LIN {X 0,Y 523.996,Z 356.21,A -85,B 0,C 180,E1 -4869.262,E2 -4869.262} C_VEL
LIN {X 0,Y 523.999,Z 356.208,A -85,B 0,C 180,E1 -4871.743,E2 -4871.743} C_VEL
LIN {X 0,Y 523.985,Z 356.213,A -85,B 0,C 180,E1 -4875.053,E2 -4875.053} C_VEL
LIN {X 0,Y 523.956,Z 356.215,A -85,B 0,C 180,E1 -4877.97,E2 -4877.97} C_VEL
LIN {X 0,Y 523.965,Z 356.22,A -85,B 0,C 180,E1 -4880.411,E2 -4880.411} C_VEL
LIN {X 0,Y 523.909,Z 356.222,A -85,B 0,C 180,E1 -4882.894,E2 -4882.894} C_VEL
LIN {X 0,Y 523.948,Z 356.211,A -85,B 0,C 180,E1 -4885.419,E2 -4885.419} C_VEL
LIN {X 0,Y 523.964,Z 356.214,A -85,B 0,C 180,E1 -4888,E2 -4888} C_VEL
LIN {X 0,Y 523.941,Z 356.216,A -85,B 0,C 180,E1 -4890.856,E2 -4890.856} C_VEL
LIN {X 0,Y 523.956,Z 356.217,A -85,B 0,C 180,E1 -4893.736,E2 -4893.736} C_VEL
LIN {X 0,Y 523.918,Z 356.224,A -85,B 0,C 180,E1 -4896.405,E2 -4896.405} C_VEL
LIN {X 0,Y 523.928,Z 356.218,A -85,B 0,C 180,E1 -4899.085,E2 -4899.085} C_VEL
LIN {X 0,Y 523.955,Z 356.22,A -85,B 0,C 180,E1 -4902.119,E2 -4902.119} C_VEL
LIN {X 0,Y 523.954,Z 356.218,A -85,B 0,C 180,E1 -4905.31,E2 -4905.31} C_VEL
LIN {X 0,Y 523.917,Z 356.22,A -85,B 0,C 180,E1 -4906.929,E2 -4906.929} C_VEL
LIN {X 0,Y 523.255,Z 356.309,A -85,B 0,C 180,E1 -4907.571,E2 -4907.571} C_VEL
LIN {X 0,Y 520.421,Z 356.663,A -85,B 0,C 180,E1 -4908.613,E2 -4908.613} C_VEL
LIN {X 0,Y 518.025,Z 356.962,A -85,B 0,C 180,E1 -4909.452,E2 -4909.452} C_VEL
LIN {X 0,Y 516.995,Z 357.088,A -85,B 0,C 180,E1 -4910.1,E2 -4910.1} C_VEL
LIN {X 0,Y 516.91,Z 357.096,A -85,B 0,C 180,E1 -4910.319,E2 -4910.319} C_VEL
LIN {X 0,Y 516.886,Z 357.099,A -85,B 0,C 180,E1 -4913.343,E2 -4913.343} C_VEL
LIN {X 0,Y 516.914,Z 357.096,A -85,B 0,C 180,E1 -4916.122,E2 -4916.122} C_VEL
LIN {X 0,Y 516.895,Z 357.097,A -85,B 0,C 180,E1 -4918.936,E2 -4918.936} C_VEL
LIN {X 0,Y 516.964,Z 357.229,A -85,B 0,C 180,E1 -4921.72,E2 -4921.72} C_VEL
LIN {X 0,Y 517.544,Z 361.865,A -85,B 0,C 180,E1 -4922.723,E2 -4922.723} C_VEL
LIN {X 0,Y 517.255,Z 376.152,A -85,B 0,C 180,E1 -4925.684,E2 -4925.684} C_VEL
LIN {X 0,Y 519.157,Z 386.668,A -85,B 0,C 180,E1 -4925.908,E2 -4925.908} C_VEL
LIN {X 0,Y 518.645,Z 483.005,A -85,B 0,C 180,E1 -4927.268,E2 -4927.268} C_VEL
LIN {X 0,Y 518.448,Z 496.309,A -85,B 0,C 180,E1 -4927.622,E2 -4927.622} C_VEL
LIN {X 0,Y 518.206,Z 508.549,A -85,B 0,C 180,E1 -4928.102,E2 -4928.102} C_VEL
LIN {X 0,Y 517.961,Z 520.129,A -85,B 0,C 180,E1 -4928.718,E2 -4928.718} C_VEL
LIN {X 0,Y 517.632,Z 531.892,A -85,B 0,C 180,E1 -4929.527,E2 -4929.527} C_VEL
LIN {X 0,Y 517.298,Z 542.625,A -85,B 0,C 180,E1 -4930.455,E2 -4930.455} C_VEL
LIN {X 0,Y 517.062,Z 551.21,A -85,B 0,C 180,E1 -4931.373,E2 -4931.373} C_VEL
LIN {X 0,Y 516.772,Z 560.444,A -85,B 0,C 180,E1 -4932.591,E2 -4932.591} C_VEL
LIN {X 0,Y 516.587,Z 567.819,A -85,B 0,C 180,E1 -4933.806,E2 -4933.806} C_VEL
LIN {X 0,Y 516.47,Z 573.778,A -85,B 0,C 180,E1 -4935.052,E2 -4935.052} C_VEL
LIN {X 0,Y 516.356,Z 578.16,A -85,B 0,C 180,E1 -4936.221,E2 -4936.221} C_VEL
LIN {X 0,Y 516.293,Z 581.562,A -85,B 0,C 180,E1 -4937.421,E2 -4937.421} C_VEL
LIN {X 0,Y 516.286,Z 583.847,A -85,B 0,C 180,E1 -4938.556,E2 -4938.556} C_VEL
LIN {X 0,Y 516.24,Z 585.354,A -85,B 0,C 180,E1 -4939.806,E2 -4939.806} C_VEL
LIN {X 0,Y 516.231,Z 585.782,A -85,B 0,C 180,E1 -4941.388,E2 -4941.388} C_VEL
LIN {X 0,Y 516.273,Z 585.416,A -85,B 0,C 180,E1 -4942.176,E2 -4942.176} C_VEL
LIN {X 0,Y 516.321,Z 583.816,A -85,B 0,C 180,E1 -4943.546,E2 -4943.546} C_VEL
LIN {X 0,Y 516.321,Z 581.857,A -85,B 0,C 180,E1 -4944.533,E2 -4944.533} C_VEL
LIN {X 0,Y 516.358,Z 578.657,A -85,B 0,C 180,E1 -4945.707,E2 -4945.707} C_VEL
LIN {X 0,Y 516.434,Z 574.411,A -85,B 0,C 180,E1 -4946.88,E2 -4946.88} C_VEL
LIN {X 0,Y 516.56,Z 568.007,A -85,B 0,C 180,E1 -4948.246,E2 -4948.246} C_VEL
LIN {X 0,Y 516.803,Z 560.982,A -85,B 0,C 180,E1 -4949.416,E2 -4949.416} C_VEL
LIN {X 0,Y 517.029,Z 552.275,A -85,B 0,C 180,E1 -4950.584,E2 -4950.584} C_VEL
LIN {X 0,Y 517.302,Z 542.393,A -85,B 0,C 180,E1 -4951.654,E2 -4951.654} C_VEL
LIN {X 0,Y 517.551,Z 532.316,A -85,B 0,C 180,E1 -4952.529,E2 -4952.529} C_VEL
LIN {X 0,Y 517.839,Z 521.167,A -85,B 0,C 180,E1 -4953.307,E2 -4953.307} C_VEL
LIN {X 0,Y 518.093,Z 509.628,A -85,B 0,C 180,E1 -4953.938,E2 -4953.938} C_VEL
LIN {X 0,Y 518.351,Z 497.014,A -85,B 0,C 180,E1 -4954.447,E2 -4954.447} C_VEL
LIN {X 0,Y 518.554,Z 483.6,A -85,B 0,C 180,E1 -4954.81,E2 -4954.81} C_VEL
LIN {X 0,Y 518.792,Z 443.561,A -85,B 0,C 180,E1 -4955.393,E2 -4955.393} C_VEL
LIN {X 0,Y 519.07,Z 385.353,A -85,B 0,C 180,E1 -4956.203,E2 -4956.203} C_VEL
LIN {X 0,Y 517.301,Z 376.098,A -85,B 0,C 180,E1 -4956.408,E2 -4956.408} C_VEL
LIN {X 0,Y 517.525,Z 361.723,A -85,B 0,C 180,E1 -4959.379,E2 -4959.379} C_VEL
LIN {X 0,Y 516.973,Z 357.093,A -85,B 0,C 180,E1 -4960.426,E2 -4960.426} C_VEL
LIN {X 0,Y 516.923,Z 357.092,A -85,B 0,C 180,E1 -4963.363,E2 -4963.363} C_VEL
LIN {X 0,Y 516.908,Z 357.093,A -85,B 0,C 180,E1 -4965.778,E2 -4965.778} C_VEL
LIN {X 0,Y 516.93,Z 357.096,A -85,B 0,C 180,E1 -4968.222,E2 -4968.222} C_VEL
LIN {X 0,Y 516.917,Z 357.094,A -85,B 0,C 180,E1 -4970.701,E2 -4970.701} C_VEL
LIN {X 0,Y 516.916,Z 357.097,A -85,B 0,C 180,E1 -4974.071,E2 -4974.071} C_VEL
LIN {X 0,Y 516.93,Z 357.092,A -85,B 0,C 180,E1 -4976.657,E2 -4976.657} C_VEL
LIN {X 0,Y 516.928,Z 357.092,A -85,B 0,C 180,E1 -4979.526,E2 -4979.526} C_VEL
LIN {X 0,Y 516.899,Z 357.096,A -85,B 0,C 180,E1 -4982.543,E2 -4982.543} C_VEL
LIN {X 0,Y 516.884,Z 357.097,A -85,B 0,C 180,E1 -4985.331,E2 -4985.331} C_VEL
LIN {X 0,Y 516.882,Z 357.102,A -85,B 0,C 180,E1 -4987.942,E2 -4987.942} C_VEL
LIN {X 0,Y 516.883,Z 357.096,A -85,B 0,C 180,E1 -4990.741,E2 -4990.741} C_VEL
LIN {X 0,Y 516.882,Z 357.096,A -85,B 0,C 180,E1 -4992.83,E2 -4992.83} C_VEL
LIN {X 0,Y 516.92,Z 357.092,A -85,B 0,C 180,E1 -4995.009,E2 -4995.009} C_VEL
LIN {X 0,Y 516.92,Z 357.093,A -85,B 0,C 180,E1 -4998.397,E2 -4998.397} C_VEL
LIN {X 0,Y 516.882,Z 357.1,A -85,B 0,C 180,E1 -5001.284,E2 -5001.284} C_VEL
LIN {X 0,Y 516.883,Z 357.099,A -85,B 0,C 180,E1 -5004.22,E2 -5004.22} C_VEL
LIN {X 0,Y 516.892,Z 357.097,A -85,B 0,C 180,E1 -5007.052,E2 -5007.052} C_VEL
LIN {X 0,Y 516.886,Z 357.102,A -85,B 0,C 180,E1 -5009.795,E2 -5009.795} C_VEL
LIN {X 0,Y 516.924,Z 357.092,A -85,B 0,C 180,E1 -5012.467,E2 -5012.467} C_VEL
LIN {X 0,Y 516.907,Z 357.097,A -85,B 0,C 180,E1 -5015.071,E2 -5015.071} C_VEL
LIN {X 0,Y 516.905,Z 357.1,A -85,B 0,C 180,E1 -5017.623,E2 -5017.623} C_VEL
LIN {X 0,Y 516.925,Z 357.092,A -85,B 0,C 180,E1 -5020.129,E2 -5020.129} C_VEL
LIN {X 0,Y 516.924,Z 357.092,A -85,B 0,C 180,E1 -5022.596,E2 -5022.596} C_VEL
LIN {X 0,Y 516.942,Z 357.094,A -85,B 0,C 180,E1 -5025.03,E2 -5025.03} C_VEL
LIN {X 0,Y 516.995,Z 357.083,A -85,B 0,C 180,E1 -5028.234,E2 -5028.234} C_VEL
LIN {X 0,Y 516.964,Z 357.092,A -85,B 0,C 180,E1 -5031.399,E2 -5031.399} C_VEL
LIN {X 0,Y 517.002,Z 357.083,A -85,B 0,C 180,E1 -5033.756,E2 -5033.756} C_VEL
LIN {X 0,Y 517.01,Z 357.086,A -85,B 0,C 180,E1 -5036.883,E2 -5036.883} C_VEL
LIN {X 0,Y 517.075,Z 357.073,A -85,B 0,C 180,E1 -5040,E2 -5040} C_VEL
LIN {X 0,Y 517.01,Z 357.086,A -85,B 0,C 180,E1 -5043.117,E2 -5043.117} C_VEL
LIN {X 0,Y 517.002,Z 357.083,A -85,B 0,C 180,E1 -5046.243,E2 -5046.243} C_VEL
LIN {X 0,Y 516.95,Z 357.09,A -85,B 0,C 180,E1 -5049.389,E2 -5049.389} C_VEL
LIN {X 0,Y 516.974,Z 357.086,A -85,B 0,C 180,E1 -5051.824,E2 -5051.824} C_VEL
LIN {X 0,Y 516.937,Z 357.093,A -85,B 0,C 180,E1 -5055.148,E2 -5055.148} C_VEL
LIN {X 0,Y 516.917,Z 357.095,A -85,B 0,C 180,E1 -5058.222,E2 -5058.222} C_VEL
LIN {X 0,Y 516.906,Z 357.099,A -85,B 0,C 180,E1 -5060.702,E2 -5060.702} C_VEL
LIN {X 0,Y 516.883,Z 357.098,A -85,B 0,C 180,E1 -5063.223,E2 -5063.223} C_VEL
LIN {X 0,Y 516.936,Z 357.094,A -85,B 0,C 180,E1 -5066.197,E2 -5066.197} C_VEL
LIN {X 0,Y 516.914,Z 357.093,A -85,B 0,C 180,E1 -5069.305,E2 -5069.305} C_VEL
LIN {X 0,Y 516.894,Z 357.1,A -85,B 0,C 180,E1 -5072.545,E2 -5072.545} C_VEL
LIN {X 0,Y 516.877,Z 357.097,A -85,B 0,C 180,E1 -5075.333,E2 -5075.333} C_VEL
LIN {X 0,Y 516.876,Z 357.101,A -85,B 0,C 180,E1 -5077.944,E2 -5077.944} C_VEL
LIN {X 0,Y 516.899,Z 357.097,A -85,B 0,C 180,E1 -5080.74,E2 -5080.74} C_VEL
LIN {X 0,Y 516.878,Z 357.101,A -85,B 0,C 180,E1 -5083.904,E2 -5083.904} C_VEL
LIN {X 0,Y 516.878,Z 357.104,A -85,B 0,C 180,E1 -5086.108,E2 -5086.108} C_VEL
LIN {X 0,Y 516.913,Z 357.096,A -85,B 0,C 180,E1 -5088.399,E2 -5088.399} C_VEL
LIN {X 0,Y 516.88,Z 357.096,A -85,B 0,C 180,E1 -5091.285,E2 -5091.285} C_VEL
LIN {X 0,Y 516.889,Z 357.1,A -85,B 0,C 180,E1 -5094.222,E2 -5094.222} C_VEL
LIN {X 0,Y 516.897,Z 357.094,A -85,B 0,C 180,E1 -5097.054,E2 -5097.054} C_VEL
LIN {X 0,Y 516.902,Z 357.1,A -85,B 0,C 180,E1 -5099.798,E2 -5099.798} C_VEL
LIN {X 0,Y 516.929,Z 357.094,A -85,B 0,C 180,E1 -5102.468,E2 -5102.468} C_VEL
LIN {X 0,Y 516.969,Z 357.23,A -85,B 0,C 180,E1 -5104.753,E2 -5104.753} C_VEL
LIN {X 0,Y 518.627,Z 366.071,A -85,B 0,C 180,E1 -5106.226,E2 -5106.226} C_VEL
LIN {X 0,Y 518.217,Z 383.586,A -85,B 0,C 180,E1 -5108.938,E2 -5108.938} C_VEL
LIN {X 0,Y 517.667,Z 405.251,A -85,B 0,C 180,E1 -5112.239,E2 -5112.239} C_VEL
LIN {X 0,Y 517.338,Z 421.391,A -85,B 0,C 180,E1 -5114.634,E2 -5114.634} C_VEL
LIN {X 0,Y 519.105,Z 433.695,A -85,B 0,C 180,E1 -5114.86,E2 -5114.86} C_VEL
LIN {X 0,Y 518.651,Z 529.669,A -85,B 0,C 180,E1 -5116.208,E2 -5116.208} C_VEL
LIN {X 0,Y 518.369,Z 542.982,A -85,B 0,C 180,E1 -5116.55,E2 -5116.55} C_VEL
LIN {X 0,Y 518.065,Z 556.304,A -85,B 0,C 180,E1 -5117.066,E2 -5117.066} C_VEL
LIN {X 0,Y 517.745,Z 568.719,A -85,B 0,C 180,E1 -5117.733,E2 -5117.733} C_VEL
LIN {X 0,Y 517.479,Z 580.42,A -85,B 0,C 180,E1 -5118.544,E2 -5118.544} C_VEL
LIN {X 0,Y 517.163,Z 590.646,A -85,B 0,C 180,E1 -5119.429,E2 -5119.429} C_VEL
LIN {X 0,Y 516.901,Z 599.85,A -85,B 0,C 180,E1 -5120.413,E2 -5120.413} C_VEL
LIN {X 0,Y 516.667,Z 608.821,A -85,B 0,C 180,E1 -5121.592,E2 -5121.592} C_VEL
LIN {X 0,Y 516.509,Z 616.045,A -85,B 0,C 180,E1 -5122.77,E2 -5122.77} C_VEL
LIN {X 0,Y 516.423,Z 622.626,A -85,B 0,C 180,E1 -5124.142,E2 -5124.142} C_VEL
LIN {X 0,Y 516.271,Z 626.976,A -85,B 0,C 180,E1 -5125.315,E2 -5125.315} C_VEL
LIN {X 0,Y 516.37,Z 629.286,A -85,B 0,C 180,E1 -5126.098,E2 -5126.098} C_VEL
LIN {X 0,Y 516.282,Z 631.151,A -85,B 0,C 180,E1 -5126.879,E2 -5126.879} C_VEL
LIN {X 0,Y 516.26,Z 632.552,A -85,B 0,C 180,E1 -5127.659,E2 -5127.659} C_VEL
LIN {X 0,Y 516.16,Z 634.157,A -85,B 0,C 180,E1 -5129.22,E2 -5129.22} C_VEL
LIN {X 0,Y 516.158,Z 634.374,A -85,B 0,C 180,E1 -5130,E2 -5130} C_VEL
LIN {X 0,Y 516.192,Z 633.548,A -85,B 0,C 180,E1 -5131.56,E2 -5131.56} C_VEL
LIN {X 0,Y 516.26,Z 632.551,A -85,B 0,C 180,E1 -5132.341,E2 -5132.341} C_VEL
LIN {X 0,Y 516.282,Z 631.149,A -85,B 0,C 180,E1 -5133.121,E2 -5133.121} C_VEL
LIN {X 0,Y 516.313,Z 628.201,A -85,B 0,C 180,E1 -5134.293,E2 -5134.293} C_VEL
LIN {X 0,Y 516.376,Z 624.212,A -85,B 0,C 180,E1 -5135.467,E2 -5135.467} C_VEL
LIN {X 0,Y 516.474,Z 618.319,A -85,B 0,C 180,E1 -5136.791,E2 -5136.791} C_VEL
LIN {X 0,Y 516.606,Z 611.374,A -85,B 0,C 180,E1 -5138.015,E2 -5138.015} C_VEL
LIN {X 0,Y 516.798,Z 603.059,A -85,B 0,C 180,E1 -5139.194,E2 -5139.194} C_VEL
LIN {X 0,Y 517.056,Z 594.541,A -85,B 0,C 180,E1 -5140.177,E2 -5140.177} C_VEL
LIN {X 0,Y 517.376,Z 584.021,A -85,B 0,C 180,E1 -5141.161,E2 -5141.161} C_VEL
LIN {X 0,Y 517.655,Z 572.813,A -85,B 0,C 180,E1 -5142.004,E2 -5142.004} C_VEL
LIN {X 0,Y 517.958,Z 562.213,A -85,B 0,C 180,E1 -5142.638,E2 -5142.638} C_VEL
LIN {X 0,Y 518.209,Z 550.516,A -85,B 0,C 180,E1 -5143.18,E2 -5143.18} C_VEL
LIN {X 0,Y 518.473,Z 537.963,A -85,B 0,C 180,E1 -5143.597,E2 -5143.597} C_VEL
LIN {X 0,Y 518.684,Z 525.252,A -85,B 0,C 180,E1 -5143.866,E2 -5143.866} C_VEL
LIN {X 0,Y 518.996,Z 432.253,A -85,B 0,C 180,E1 -5145.163,E2 -5145.163} C_VEL
LIN {X 0,Y 517.327,Z 421.066,A -85,B 0,C 180,E1 -5145.377,E2 -5145.377} C_VEL
LIN {X 0,Y 517.765,Z 399.658,A -85,B 0,C 180,E1 -5148.601,E2 -5148.601} C_VEL
LIN {X 0,Y 518.262,Z 380.796,A -85,B 0,C 180,E1 -5151.477,E2 -5151.477} C_VEL
LIN {X 0,Y 518.645,Z 366,A -85,B 0,C 180,E1 -5153.774,E2 -5153.774} C_VEL
LIN {X 0,Y 516.951,Z 357.093,A -85,B 0,C 180,E1 -5155.302,E2 -5155.302} C_VEL
LIN {X 0,Y 516.925,Z 357.096,A -85,B 0,C 180,E1 -5158.414,E2 -5158.414} C_VEL
LIN {X 0,Y 516.891,Z 357.093,A -85,B 0,C 180,E1 -5161.109,E2 -5161.109} C_VEL
LIN {X 0,Y 516.911,Z 357.1,A -85,B 0,C 180,E1 -5163.966,E2 -5163.966} C_VEL
LIN {X 0,Y 516.881,Z 357.097,A -85,B 0,C 180,E1 -5166.745,E2 -5166.745} C_VEL
LIN {X 0,Y 516.879,Z 357.102,A -85,B 0,C 180,E1 -5169.72,E2 -5169.72} C_VEL
LIN {X 0,Y 516.912,Z 357.099,A -85,B 0,C 180,E1 -5171.774,E2 -5171.774} C_VEL
LIN {X 0,Y 516.918,Z 357.09,A -85,B 0,C 180,E1 -5175.009,E2 -5175.009} C_VEL
LIN {X 0,Y 516.917,Z 357.09,A -85,B 0,C 180,E1 -5178.397,E2 -5178.397} C_VEL
LIN {X 0,Y 516.881,Z 357.098,A -85,B 0,C 180,E1 -5181.284,E2 -5181.284} C_VEL
LIN {X 0,Y 516.886,Z 357.095,A -85,B 0,C 180,E1 -5184.221,E2 -5184.221} C_VEL
LIN {X 0,Y 516.892,Z 357.097,A -85,B 0,C 180,E1 -5187.053,E2 -5187.053} C_VEL
LIN {X 0,Y 516.895,Z 357.097,A -85,B 0,C 180,E1 -5189.796,E2 -5189.796} C_VEL
LIN {X 0,Y 516.922,Z 357.09,A -85,B 0,C 180,E1 -5192.467,E2 -5192.467} C_VEL
LIN {X 0,Y 516.906,Z 357.091,A -85,B 0,C 180,E1 -5195.072,E2 -5195.072} C_VEL
LIN {X 0,Y 516.904,Z 357.097,A -85,B 0,C 180,E1 -5197.623,E2 -5197.623} C_VEL
LIN {X 0,Y 516.924,Z 357.089,A -85,B 0,C 180,E1 -5200.13,E2 -5200.13} C_VEL
LIN {X 0,Y 516.923,Z 357.091,A -85,B 0,C 180,E1 -5202.596,E2 -5202.596} C_VEL
LIN {X 0,Y 516.932,Z 357.095,A -85,B 0,C 180,E1 -5205.03,E2 -5205.03} C_VEL
LIN {X 0,Y 516.994,Z 357.081,A -85,B 0,C 180,E1 -5208.234,E2 -5208.234} C_VEL
LIN {X 0,Y 516.965,Z 357.089,A -85,B 0,C 180,E1 -5211.4,E2 -5211.4} C_VEL
LIN {X 0,Y 517.002,Z 357.078,A -85,B 0,C 180,E1 -5213.757,E2 -5213.757} C_VEL
LIN {X 0,Y 517.011,Z 357.088,A -85,B 0,C 180,E1 -5216.883,E2 -5216.883} C_VEL
LIN {X 0,Y 517.075,Z 357.07,A -85,B 0,C 180,E1 -5220,E2 -5220} C_VEL
LIN {X 0,Y 517.01,Z 357.081,A -85,B 0,C 180,E1 -5223.117,E2 -5223.117} C_VEL
LIN {X 0,Y 517.002,Z 357.083,A -85,B 0,C 180,E1 -5226.244,E2 -5226.244} C_VEL
LIN {X 0,Y 516.95,Z 357.087,A -85,B 0,C 180,E1 -5229.39,E2 -5229.39} C_VEL
LIN {X 0,Y 516.948,Z 357.087,A -85,B 0,C 180,E1 -5231.811,E2 -5231.811} C_VEL
LIN {X 0,Y 516.938,Z 357.09,A -85,B 0,C 180,E1 -5235.148,E2 -5235.148} C_VEL
LIN {X 0,Y 516.918,Z 357.094,A -85,B 0,C 180,E1 -5238.223,E2 -5238.223} C_VEL
LIN {X 0,Y 516.905,Z 357.096,A -85,B 0,C 180,E1 -5240.702,E2 -5240.702} C_VEL
LIN {X 0,Y 516.904,Z 357.097,A -85,B 0,C 180,E1 -5244.073,E2 -5244.073} C_VEL
LIN {X 0,Y 516.922,Z 357.09,A -85,B 0,C 180,E1 -5246.658,E2 -5246.658} C_VEL
LIN {X 0,Y 516.905,Z 357.093,A -85,B 0,C 180,E1 -5249.525,E2 -5249.525} C_VEL
LIN {X 0,Y 516.895,Z 357.098,A -85,B 0,C 180,E1 -5252.545,E2 -5252.545} C_VEL
LIN {X 0,Y 516.878,Z 357.097,A -85,B 0,C 180,E1 -5255.333,E2 -5255.333} C_VEL
LIN {X 0,Y 516.878,Z 357.103,A -85,B 0,C 180,E1 -5257.944,E2 -5257.944} C_VEL
LIN {X 0,Y 516.901,Z 357.095,A -85,B 0,C 180,E1 -5260.741,E2 -5260.741} C_VEL
LIN {X 0,Y 516.88,Z 357.104,A -85,B 0,C 180,E1 -5263.904,E2 -5263.904} C_VEL
LIN {X 0,Y 516.88,Z 357.102,A -85,B 0,C 180,E1 -5266.108,E2 -5266.108} C_VEL
LIN {X 0,Y 516.904,Z 357.096,A -85,B 0,C 180,E1 -5269.261,E2 -5269.261} C_VEL
LIN {X 0,Y 516.91,Z 357.096,A -85,B 0,C 180,E1 -5270.319,E2 -5270.319} C_VEL
LIN {X 0,Y 516.242,Z 357.177,A -85,B 0,C 180,E1 -5270.969,E2 -5270.969} C_VEL
LIN {X 0,Y 513.384,Z 357.538,A -85,B 0,C 180,E1 -5272.025,E2 -5272.025} C_VEL
LIN {X 0,Y 510.965,Z 357.842,A -85,B 0,C 180,E1 -5272.875,E2 -5272.875} C_VEL
LIN {X 0,Y 509.92,Z 357.97,A -85,B 0,C 180,E1 -5273.531,E2 -5273.531} C_VEL
LIN {X 0,Y 509.832,Z 357.979,A -85,B 0,C 180,E1 -5273.753,E2 -5273.753} C_VEL
LIN {X 0,Y 509.864,Z 357.971,A -85,B 0,C 180,E1 -5276.54,E2 -5276.54} C_VEL
LIN {X 0,Y 509.852,Z 357.978,A -85,B 0,C 180,E1 -5279.335,E2 -5279.335} C_VEL
LIN {X 0,Y 509.904,Z 358.006,A -85,B 0,C 180,E1 -5281.549,E2 -5281.549} C_VEL
LIN {X 0,Y 510.582,Z 363.554,A -85,B 0,C 180,E1 -5282.763,E2 -5282.763} C_VEL
LIN {X 0,Y 510.28,Z 376.526,A -85,B 0,C 180,E1 -5285.479,E2 -5285.479} C_VEL
LIN {X 0,Y 512.342,Z 387.866,A -85,B 0,C 180,E1 -5285.714,E2 -5285.714} C_VEL
LIN {X 0,Y 511.762,Z 482.882,A -85,B 0,C 180,E1 -5287.069,E2 -5287.069} C_VEL
LIN {X 0,Y 511.58,Z 495.634,A -85,B 0,C 180,E1 -5287.405,E2 -5287.405} C_VEL
LIN {X 0,Y 511.321,Z 508.278,A -85,B 0,C 180,E1 -5287.898,E2 -5287.898} C_VEL
LIN {X 0,Y 511.046,Z 520.038,A -85,B 0,C 180,E1 -5288.522,E2 -5288.522} C_VEL
LIN {X 0,Y 510.736,Z 530.852,A -85,B 0,C 180,E1 -5289.262,E2 -5289.262} C_VEL
LIN {X 0,Y 510.372,Z 541.584,A -85,B 0,C 180,E1 -5290.179,E2 -5290.179} C_VEL
LIN {X 0,Y 510.109,Z 550.431,A -85,B 0,C 180,E1 -5291.109,E2 -5291.109} C_VEL
LIN {X 0,Y 509.832,Z 558.487,A -85,B 0,C 180,E1 -5292.137,E2 -5292.137} C_VEL
LIN {X 0,Y 509.629,Z 566.3,A -85,B 0,C 180,E1 -5293.373,E2 -5293.373} C_VEL
LIN {X 0,Y 509.46,Z 571.581,A -85,B 0,C 180,E1 -5294.395,E2 -5294.395} C_VEL
LIN {X 0,Y 509.327,Z 576.648,A -85,B 0,C 180,E1 -5295.619,E2 -5295.619} C_VEL
LIN {X 0,Y 509.243,Z 580.53,A -85,B 0,C 180,E1 -5296.838,E2 -5296.838} C_VEL
LIN {X 0,Y 509.212,Z 584.15,A -85,B 0,C 180,E1 -5298.502,E2 -5298.502} C_VEL
LIN {X 0,Y 509.178,Z 585.572,A -85,B 0,C 180,E1 -5299.663,E2 -5299.663} C_VEL
LIN {X 0,Y 509.094,Z 586.073,A -85,B 0,C 180,E1 -5300.465,E2 -5300.465} C_VEL
LIN {X 0,Y 509.177,Z 585.824,A -85,B 0,C 180,E1 -5302.067,E2 -5302.067} C_VEL
LIN {X 0,Y 509.243,Z 584.192,A -85,B 0,C 180,E1 -5303.552,E2 -5303.552} C_VEL
LIN {X 0,Y 509.249,Z 582.466,A -85,B 0,C 180,E1 -5304.456,E2 -5304.456} C_VEL
LIN {X 0,Y 509.28,Z 579.374,A -85,B 0,C 180,E1 -5305.647,E2 -5305.647} C_VEL
LIN {X 0,Y 509.372,Z 575.24,A -85,B 0,C 180,E1 -5306.836,E2 -5306.836} C_VEL
LIN {X 0,Y 509.474,Z 568.968,A -85,B 0,C 180,E1 -5308.221,E2 -5308.221} C_VEL
LIN {X 0,Y 509.749,Z 562.134,A -85,B 0,C 180,E1 -5309.408,E2 -5309.408} C_VEL
LIN {X 0,Y 510.006,Z 553.606,A -85,B 0,C 180,E1 -5310.592,E2 -5310.592} C_VEL
LIN {X 0,Y 510.282,Z 544.894,A -85,B 0,C 180,E1 -5311.578,E2 -5311.578} C_VEL
LIN {X 0,Y 510.533,Z 534.214,A -85,B 0,C 180,E1 -5312.564,E2 -5312.564} C_VEL
LIN {X 0,Y 510.901,Z 523.424,A -85,B 0,C 180,E1 -5313.352,E2 -5313.352} C_VEL
LIN {X 0,Y 511.174,Z 511.41,A -85,B 0,C 180,E1 -5314.04,E2 -5314.04} C_VEL
LIN {X 0,Y 511.43,Z 498.807,A -85,B 0,C 180,E1 -5314.581,E2 -5314.581} C_VEL
LIN {X 0,Y 511.655,Z 486.163,A -85,B 0,C 180,E1 -5314.949,E2 -5314.949} C_VEL
LIN {X 0,Y 511.761,Z 468.451,A -85,B 0,C 180,E1 -5315.245,E2 -5315.245} C_VEL
LIN {X 0,Y 512.267,Z 386.422,A -85,B 0,C 180,E1 -5316.399,E2 -5316.399} C_VEL
LIN {X 0,Y 510.328,Z 376.422,A -85,B 0,C 180,E1 -5316.619,E2 -5316.619} C_VEL
LIN {X 0,Y 510.531,Z 362.613,A -85,B 0,C 180,E1 -5319.508,E2 -5319.508} C_VEL
LIN {X 0,Y 509.92,Z 357.971,A -85,B 0,C 180,E1 -5320.572,E2 -5320.572} C_VEL
LIN {X 0,Y 509.868,Z 357.971,A -85,B 0,C 180,E1 -5323.552,E2 -5323.552} C_VEL
LIN {X 0,Y 509.861,Z 357.975,A -85,B 0,C 180,E1 -5326.002,E2 -5326.002} C_VEL
LIN {X 0,Y 509.871,Z 357.975,A -85,B 0,C 180,E1 -5328.483,E2 -5328.483} C_VEL
LIN {X 0,Y 509.855,Z 357.972,A -85,B 0,C 180,E1 -5331.001,E2 -5331.001} C_VEL
LIN {X 0,Y 509.841,Z 357.974,A -85,B 0,C 180,E1 -5333.562,E2 -5333.562} C_VEL
LIN {X 0,Y 509.915,Z 357.97,A -85,B 0,C 180,E1 -5336.378,E2 -5336.378} C_VEL
LIN {X 0,Y 509.889,Z 357.968,A -85,B 0,C 180,E1 -5338.843,E2 -5338.843} C_VEL
LIN {X 0,Y 509.824,Z 357.978,A -85,B 0,C 180,E1 -5341.589,E2 -5341.589} C_VEL
LIN {X 0,Y 509.855,Z 357.975,A -85,B 0,C 180,E1 -5344.412,E2 -5344.412} C_VEL
LIN {X 0,Y 509.82,Z 357.977,A -85,B 0,C 180,E1 -5347.34,E2 -5347.34} C_VEL
LIN {X 0,Y 509.837,Z 357.977,A -85,B 0,C 180,E1 -5350.381,E2 -5350.381} C_VEL
LIN {X 0,Y 509.822,Z 357.976,A -85,B 0,C 180,E1 -5353.061,E2 -5353.061} C_VEL
LIN {X 0,Y 509.829,Z 357.98,A -85,B 0,C 180,E1 -5355.791,E2 -5355.791} C_VEL
LIN {X 0,Y 509.863,Z 357.972,A -85,B 0,C 180,E1 -5358.575,E2 -5358.575} C_VEL
LIN {X 0,Y 509.848,Z 357.979,A -85,B 0,C 180,E1 -5361.785,E2 -5361.785} C_VEL
LIN {X 0,Y 509.838,Z 357.974,A -85,B 0,C 180,E1 -5364.622,E2 -5364.622} C_VEL
LIN {X 0,Y 509.86,Z 357.976,A -85,B 0,C 180,E1 -5367.48,E2 -5367.48} C_VEL
LIN {X 0,Y 509.852,Z 357.974,A -85,B 0,C 180,E1 -5370.273,E2 -5370.273} C_VEL
LIN {X 0,Y 509.881,Z 357.971,A -85,B 0,C 180,E1 -5372.944,E2 -5372.944} C_VEL
LIN {X 0,Y 509.869,Z 357.976,A -85,B 0,C 180,E1 -5375.574,E2 -5375.574} C_VEL
LIN {X 0,Y 509.842,Z 357.975,A -85,B 0,C 180,E1 -5378.149,E2 -5378.149} C_VEL
LIN {X 0,Y 509.858,Z 357.973,A -85,B 0,C 180,E1 -5380.681,E2 -5380.681} C_VEL
LIN {X 0,Y 509.88,Z 357.974,A -85,B 0,C 180,E1 -5383.174,E2 -5383.174} C_VEL
LIN {X 0,Y 509.865,Z 357.975,A -85,B 0,C 180,E1 -5385.634,E2 -5385.634} C_VEL
LIN {X 0,Y 509.917,Z 357.969,A -85,B 0,C 180,E1 -5388.874,E2 -5388.874} C_VEL
LIN {X 0,Y 509.943,Z 357.962,A -85,B 0,C 180,E1 -5392.078,E2 -5392.078} C_VEL
LIN {X 0,Y 509.976,Z 357.959,A -85,B 0,C 180,E1 -5394.464,E2 -5394.464} C_VEL
LIN {X 0,Y 510.047,Z 357.95,A -85,B 0,C 180,E1 -5397.631,E2 -5397.631} C_VEL
LIN {X 0,Y 510.058,Z 357.952,A -85,B 0,C 180,E1 -5400.789,E2 -5400.789} C_VEL
LIN {X 0,Y 509.953,Z 357.965,A -85,B 0,C 180,E1 -5403.16,E2 -5403.16} C_VEL
LIN {X 0,Y 509.97,Z 357.96,A -85,B 0,C 180,E1 -5406.33,E2 -5406.33} C_VEL
LIN {X 0,Y 509.91,Z 357.971,A -85,B 0,C 180,E1 -5408.72,E2 -5408.72} C_VEL
LIN {X 0,Y 509.942,Z 357.962,A -85,B 0,C 180,E1 -5411.931,E2 -5411.931} C_VEL
LIN {X 0,Y 509.884,Z 357.971,A -85,B 0,C 180,E1 -5415.242,E2 -5415.242} C_VEL
LIN {X 0,Y 509.879,Z 357.97,A -85,B 0,C 180,E1 -5418.001,E2 -5418.001} C_VEL
LIN {X 0,Y 509.849,Z 357.977,A -85,B 0,C 180,E1 -5421.002,E2 -5421.002} C_VEL
LIN {X 0,Y 509.842,Z 357.974,A -85,B 0,C 180,E1 -5423.563,E2 -5423.563} C_VEL
LIN {X 0,Y 509.905,Z 357.973,A -85,B 0,C 180,E1 -5426.38,E2 -5426.38} C_VEL
LIN {X 0,Y 509.87,Z 357.974,A -85,B 0,C 180,E1 -5428.845,E2 -5428.845} C_VEL
LIN {X 0,Y 509.818,Z 357.977,A -85,B 0,C 180,E1 -5431.59,E2 -5431.59} C_VEL
LIN {X 0,Y 509.848,Z 357.978,A -85,B 0,C 180,E1 -5434.414,E2 -5434.414} C_VEL
LIN {X 0,Y 509.814,Z 357.977,A -85,B 0,C 180,E1 -5437.341,E2 -5437.341} C_VEL
LIN {X 0,Y 509.856,Z 357.977,A -85,B 0,C 180,E1 -5440.381,E2 -5440.381} C_VEL
LIN {X 0,Y 509.835,Z 357.974,A -85,B 0,C 180,E1 -5443.065,E2 -5443.065} C_VEL
LIN {X 0,Y 509.826,Z 357.979,A -85,B 0,C 180,E1 -5445.793,E2 -5445.793} C_VEL
LIN {X 0,Y 509.855,Z 357.974,A -85,B 0,C 180,E1 -5448.576,E2 -5448.576} C_VEL
LIN {X 0,Y 509.849,Z 357.977,A -85,B 0,C 180,E1 -5451.787,E2 -5451.787} C_VEL
LIN {X 0,Y 509.845,Z 357.974,A -85,B 0,C 180,E1 -5454.624,E2 -5454.624} C_VEL
LIN {X 0,Y 509.865,Z 357.972,A -85,B 0,C 180,E1 -5457.482,E2 -5457.482} C_VEL
LIN {X 0,Y 509.881,Z 357.973,A -85,B 0,C 180,E1 -5460.27,E2 -5460.27} C_VEL
LIN {X 0,Y 509.886,Z 357.97,A -85,B 0,C 180,E1 -5462.945,E2 -5462.945} C_VEL
LIN {X 0,Y 509.929,Z 358.066,A -85,B 0,C 180,E1 -5464.571,E2 -5464.571} C_VEL
LIN {X 0,Y 511.646,Z 367.113,A -85,B 0,C 180,E1 -5466.096,E2 -5466.096} C_VEL
LIN {X 0,Y 511.449,Z 377.899,A -85,B 0,C 180,E1 -5467.798,E2 -5467.798} C_VEL
LIN {X 0,Y 510.836,Z 398.069,A -85,B 0,C 180,E1 -5470.929,E2 -5470.929} C_VEL
LIN {X 0,Y 510.365,Z 416.852,A -85,B 0,C 180,E1 -5473.809,E2 -5473.809} C_VEL
LIN {X 0,Y 510.321,Z 420.828,A -85,B 0,C 180,E1 -5474.414,E2 -5474.414} C_VEL
LIN {X 0,Y 512.253,Z 435.543,A -85,B 0,C 180,E1 -5474.683,E2 -5474.683} C_VEL
LIN {X 0,Y 511.751,Z 529.318,A -85,B 0,C 180,E1 -5476.018,E2 -5476.018} C_VEL
LIN {X 0,Y 511.454,Z 542.638,A -85,B 0,C 180,E1 -5476.365,E2 -5476.365} C_VEL
LIN {X 0,Y 511.147,Z 555.965,A -85,B 0,C 180,E1 -5476.888,E2 -5476.888} C_VEL
LIN {X 0,Y 510.824,Z 567.693,A -85,B 0,C 180,E1 -5477.52,E2 -5477.52} C_VEL
LIN {X 0,Y 510.516,Z 578.785,A -85,B 0,C 180,E1 -5478.285,E2 -5478.285} C_VEL
LIN {X 0,Y 510.199,Z 589.261,A -85,B 0,C 180,E1 -5479.183,E2 -5479.183} C_VEL
LIN {X 0,Y 509.938,Z 597.83,A -85,B 0,C 180,E1 -5480.08,E2 -5480.08} C_VEL
LIN {X 0,Y 509.682,Z 605.737,A -85,B 0,C 180,E1 -5481.076,E2 -5481.076} C_VEL
LIN {X 0,Y 509.476,Z 613.463,A -85,B 0,C 180,E1 -5482.271,E2 -5482.271} C_VEL
LIN {X 0,Y 509.317,Z 619.722,A -85,B 0,C 180,E1 -5483.474,E2 -5483.474} C_VEL
LIN {X 0,Y 509.243,Z 625.327,A -85,B 0,C 180,E1 -5484.853,E2 -5484.853} C_VEL
LIN {X 0,Y 509.275,Z 628.953,A -85,B 0,C 180,E1 -5486.044,E2 -5486.044} C_VEL
LIN {X 0,Y 509.201,Z 630.819,A -85,B 0,C 180,E1 -5486.835,E2 -5486.835} C_VEL
LIN {X 0,Y 509.189,Z 632.22,A -85,B 0,C 180,E1 -5487.627,E2 -5487.627} C_VEL
LIN {X 0,Y 509.073,Z 633.824,A -85,B 0,C 180,E1 -5489.209,E2 -5489.209} C_VEL
LIN {X 0,Y 509.069,Z 634.04,A -85,B 0,C 180,E1 -5490,E2 -5490} C_VEL
LIN {X 0,Y 509.112,Z 633.214,A -85,B 0,C 180,E1 -5491.582,E2 -5491.582} C_VEL
LIN {X 0,Y 509.189,Z 632.217,A -85,B 0,C 180,E1 -5492.373,E2 -5492.373} C_VEL
LIN {X 0,Y 509.201,Z 630.814,A -85,B 0,C 180,E1 -5493.165,E2 -5493.165} C_VEL
LIN {X 0,Y 509.206,Z 627.864,A -85,B 0,C 180,E1 -5494.353,E2 -5494.353} C_VEL
LIN {X 0,Y 509.294,Z 623.874,A -85,B 0,C 180,E1 -5495.543,E2 -5495.543} C_VEL
LIN {X 0,Y 509.407,Z 617.839,A -85,B 0,C 180,E1 -5496.914,E2 -5496.914} C_VEL
LIN {X 0,Y 509.551,Z 611.032,A -85,B 0,C 180,E1 -5498.127,E2 -5498.127} C_VEL
LIN {X 0,Y 509.753,Z 602.716,A -85,B 0,C 180,E1 -5499.323,E2 -5499.323} C_VEL
LIN {X 0,Y 510.025,Z 594.197,A -85,B 0,C 180,E1 -5500.319,E2 -5500.319} C_VEL
LIN {X 0,Y 510.387,Z 583.675,A -85,B 0,C 180,E1 -5501.316,E2 -5501.316} C_VEL
LIN {X 0,Y 510.665,Z 572.465,A -85,B 0,C 180,E1 -5502.171,E2 -5502.171} C_VEL
LIN {X 0,Y 511.007,Z 561.864,A -85,B 0,C 180,E1 -5502.813,E2 -5502.813} C_VEL
LIN {X 0,Y 511.298,Z 550.164,A -85,B 0,C 180,E1 -5503.361,E2 -5503.361} C_VEL
LIN {X 0,Y 511.574,Z 537.606,A -85,B 0,C 180,E1 -5503.784,E2 -5503.784} C_VEL
LIN {X 0,Y 511.788,Z 524.885,A -85,B 0,C 180,E1 -5504.057,E2 -5504.057} C_VEL
LIN {X 0,Y 512.117,Z 432.764,A -85,B 0,C 180,E1 -5505.36,E2 -5505.36} C_VEL
LIN {X 0,Y 510.289,Z 420.651,A -85,B 0,C 180,E1 -5505.605,E2 -5505.605} C_VEL
LIN {X 0,Y 510.762,Z 400.678,A -85,B 0,C 180,E1 -5508.657,E2 -5508.657} C_VEL
LIN {X 0,Y 511.308,Z 381.857,A -85,B 0,C 180,E1 -5511.572,E2 -5511.572} C_VEL
LIN {X 0,Y 511.671,Z 367.107,A -85,B 0,C 180,E1 -5513.903,E2 -5513.903} C_VEL
LIN {X 0,Y 509.921,Z 357.97,A -85,B 0,C 180,E1 -5515.484,E2 -5515.484} C_VEL
LIN {X 0,Y 509.886,Z 357.969,A -85,B 0,C 180,E1 -5518.843,E2 -5518.843} C_VEL
LIN {X 0,Y 509.826,Z 357.976,A -85,B 0,C 180,E1 -5521.589,E2 -5521.589} C_VEL
LIN {X 0,Y 509.852,Z 357.975,A -85,B 0,C 180,E1 -5524.412,E2 -5524.412} C_VEL
LIN {X 0,Y 509.817,Z 357.978,A -85,B 0,C 180,E1 -5527.34,E2 -5527.34} C_VEL
LIN {X 0,Y 509.835,Z 357.975,A -85,B 0,C 180,E1 -5530.381,E2 -5530.381} C_VEL
LIN {X 0,Y 509.819,Z 357.975,A -85,B 0,C 180,E1 -5533.062,E2 -5533.062} C_VEL
LIN {X 0,Y 509.826,Z 357.98,A -85,B 0,C 180,E1 -5535.792,E2 -5535.792} C_VEL
LIN {X 0,Y 509.86,Z 357.969,A -85,B 0,C 180,E1 -5538.575,E2 -5538.575} C_VEL
LIN {X 0,Y 509.847,Z 357.977,A -85,B 0,C 180,E1 -5541.785,E2 -5541.785} C_VEL
LIN {X 0,Y 509.84,Z 357.972,A -85,B 0,C 180,E1 -5544.623,E2 -5544.623} C_VEL
LIN {X 0,Y 509.859,Z 357.978,A -85,B 0,C 180,E1 -5547.481,E2 -5547.481} C_VEL
LIN {X 0,Y 509.874,Z 357.968,A -85,B 0,C 180,E1 -5550.268,E2 -5550.268} C_VEL
LIN {X 0,Y 509.88,Z 357.97,A -85,B 0,C 180,E1 -5552.944,E2 -5552.944} C_VEL
LIN {X 0,Y 509.867,Z 357.969,A -85,B 0,C 180,E1 -5555.574,E2 -5555.574} C_VEL
LIN {X 0,Y 509.84,Z 357.973,A -85,B 0,C 180,E1 -5558.15,E2 -5558.15} C_VEL
LIN {X 0,Y 509.857,Z 357.971,A -85,B 0,C 180,E1 -5560.681,E2 -5560.681} C_VEL
LIN {X 0,Y 509.879,Z 357.976,A -85,B 0,C 180,E1 -5563.175,E2 -5563.175} C_VEL
LIN {X 0,Y 509.855,Z 357.972,A -85,B 0,C 180,E1 -5565.634,E2 -5565.634} C_VEL
LIN {X 0,Y 509.92,Z 357.968,A -85,B 0,C 180,E1 -5568.875,E2 -5568.875} C_VEL
LIN {X 0,Y 509.943,Z 357.96,A -85,B 0,C 180,E1 -5572.078,E2 -5572.078} C_VEL
LIN {X 0,Y 509.976,Z 357.955,A -85,B 0,C 180,E1 -5574.464,E2 -5574.464} C_VEL
LIN {X 0,Y 510.047,Z 357.946,A -85,B 0,C 180,E1 -5577.631,E2 -5577.631} C_VEL
LIN {X 0,Y 510.058,Z 357.953,A -85,B 0,C 180,E1 -5580.79,E2 -5580.79} C_VEL
LIN {X 0,Y 509.952,Z 357.96,A -85,B 0,C 180,E1 -5583.16,E2 -5583.16} C_VEL
LIN {X 0,Y 509.97,Z 357.96,A -85,B 0,C 180,E1 -5586.33,E2 -5586.33} C_VEL
LIN {X 0,Y 509.911,Z 357.97,A -85,B 0,C 180,E1 -5588.721,E2 -5588.721} C_VEL
LIN {X 0,Y 509.896,Z 357.966,A -85,B 0,C 180,E1 -5591.932,E2 -5591.932} C_VEL
LIN {X 0,Y 509.885,Z 357.968,A -85,B 0,C 180,E1 -5595.242,E2 -5595.242} C_VEL
LIN {X 0,Y 509.88,Z 357.968,A -85,B 0,C 180,E1 -5598.002,E2 -5598.002} C_VEL
LIN {X 0,Y 509.843,Z 357.973,A -85,B 0,C 180,E1 -5601.002,E2 -5601.002} C_VEL
LIN {X 0,Y 509.829,Z 357.974,A -85,B 0,C 180,E1 -5603.564,E2 -5603.564} C_VEL
LIN {X 0,Y 509.907,Z 357.964,A -85,B 0,C 180,E1 -5606.38,E2 -5606.38} C_VEL
LIN {X 0,Y 509.871,Z 357.971,A -85,B 0,C 180,E1 -5608.845,E2 -5608.845} C_VEL
LIN {X 0,Y 509.82,Z 357.975,A -85,B 0,C 180,E1 -5611.591,E2 -5611.591} C_VEL
LIN {X 0,Y 509.849,Z 357.977,A -85,B 0,C 180,E1 -5614.414,E2 -5614.414} C_VEL
LIN {X 0,Y 509.815,Z 357.976,A -85,B 0,C 180,E1 -5617.341,E2 -5617.341} C_VEL
LIN {X 0,Y 509.858,Z 357.976,A -85,B 0,C 180,E1 -5620.381,E2 -5620.381} C_VEL
LIN {X 0,Y 509.837,Z 357.973,A -85,B 0,C 180,E1 -5623.065,E2 -5623.065} C_VEL
LIN {X 0,Y 509.829,Z 357.982,A -85,B 0,C 180,E1 -5625.793,E2 -5625.793} C_VEL
LIN {X 0,Y 509.865,Z 357.973,A -85,B 0,C 180,E1 -5628.577,E2 -5628.577} C_VEL
LIN {X 0,Y 509.859,Z 357.978,A -85,B 0,C 180,E1 -5631.664,E2 -5631.664} C_VEL
LIN {X 0,Y 509.832,Z 357.979,A -85,B 0,C 180,E1 -5633.753,E2 -5633.753} C_VEL
LIN {X 0,Y 509.167,Z 358.06,A -85,B 0,C 180,E1 -5634.413,E2 -5634.413} C_VEL
LIN {X 0,Y 506.349,Z 358.414,A -85,B 0,C 180,E1 -5635.485,E2 -5635.485} C_VEL
LIN {X 0,Y 503.955,Z 358.71,A -85,B 0,C 180,E1 -5636.348,E2 -5636.348} C_VEL
LIN {X 0,Y 502.906,Z 358.839,A -85,B 0,C 180,E1 -5637.015,E2 -5637.015} C_VEL
LIN {X 0,Y 502.809,Z 358.85,A -85,B 0,C 180,E1 -5637.24,E2 -5637.24} C_VEL
LIN {X 0,Y 502.833,Z 358.852,A -85,B 0,C 180,E1 -5640.063,E2 -5640.063} C_VEL
LIN {X 0,Y 502.871,Z 358.939,A -85,B 0,C 180,E1 -5641.402,E2 -5641.402} C_VEL
LIN {X 0,Y 503.633,Z 364.22,A -85,B 0,C 180,E1 -5642.581,E2 -5642.581} C_VEL
LIN {X 0,Y 503.311,Z 376.831,A -85,B 0,C 180,E1 -5645.258,E2 -5645.258} C_VEL
LIN {X 0,Y 505.461,Z 387.84,A -85,B 0,C 180,E1 -5645.494,E2 -5645.494} C_VEL
LIN {X 0,Y 504.896,Z 482.835,A -85,B 0,C 180,E1 -5646.867,E2 -5646.867} C_VEL
LIN {X 0,Y 504.691,Z 495.935,A -85,B 0,C 180,E1 -5647.214,E2 -5647.214} C_VEL
LIN {X 0,Y 504.41,Z 509.178,A -85,B 0,C 180,E1 -5647.741,E2 -5647.741} C_VEL
LIN {X 0,Y 504.149,Z 519.937,A -85,B 0,C 180,E1 -5648.321,E2 -5648.321} C_VEL
LIN {X 0,Y 503.84,Z 530.31,A -85,B 0,C 180,E1 -5649.029,E2 -5649.029} C_VEL
LIN {X 0,Y 503.428,Z 541.635,A -85,B 0,C 180,E1 -5650,E2 -5650} C_VEL
LIN {X 0,Y 503.111,Z 551.439,A -85,B 0,C 180,E1 -5651.048,E2 -5651.048} C_VEL
LIN {X 0,Y 502.791,Z 559.367,A -85,B 0,C 180,E1 -5652.091,E2 -5652.091} C_VEL
LIN {X 0,Y 502.575,Z 567.058,A -85,B 0,C 180,E1 -5653.342,E2 -5653.342} C_VEL
LIN {X 0,Y 502.379,Z 573.179,A -85,B 0,C 180,E1 -5654.586,E2 -5654.586} C_VEL
LIN {X 0,Y 502.24,Z 577.974,A -85,B 0,C 180,E1 -5655.825,E2 -5655.825} C_VEL
LIN {X 0,Y 502.168,Z 581.604,A -85,B 0,C 180,E1 -5657.061,E2 -5657.061} C_VEL
LIN {X 0,Y 502.123,Z 584.468,A -85,B 0,C 180,E1 -5658.455,E2 -5658.455} C_VEL
LIN {X 0,Y 502.084,Z 585.78,A -85,B 0,C 180,E1 -5659.516,E2 -5659.516} C_VEL
LIN {X 0,Y 502.017,Z 586.354,A -85,B 0,C 180,E1 -5660.329,E2 -5660.329} C_VEL
LIN {X 0,Y 502.051,Z 586.5,A -85,B 0,C 180,E1 -5661.142,E2 -5661.142} C_VEL
LIN {X 0,Y 502.098,Z 586.232,A -85,B 0,C 180,E1 -5661.954,E2 -5661.954} C_VEL
LIN {X 0,Y 502.15,Z 584.547,A -85,B 0,C 180,E1 -5663.571,E2 -5663.571} C_VEL
LIN {X 0,Y 502.181,Z 583.074,A -85,B 0,C 180,E1 -5664.378,E2 -5664.378} C_VEL
LIN {X 0,Y 502.204,Z 580.091,A -85,B 0,C 180,E1 -5665.586,E2 -5665.586} C_VEL
LIN {X 0,Y 502.312,Z 576.07,A -85,B 0,C 180,E1 -5666.792,E2 -5666.792} C_VEL
LIN {X 0,Y 502.361,Z 570.92,A -85,B 0,C 180,E1 -5667.996,E2 -5667.996} C_VEL
LIN {X 0,Y 502.655,Z 564.442,A -85,B 0,C 180,E1 -5669.199,E2 -5669.199} C_VEL
LIN {X 0,Y 502.877,Z 556.437,A -85,B 0,C 180,E1 -5670.4,E2 -5670.4} C_VEL
LIN {X 0,Y 503.168,Z 548.269,A -85,B 0,C 180,E1 -5671.401,E2 -5671.401} C_VEL
LIN {X 0,Y 503.479,Z 538.291,A -85,B 0,C 180,E1 -5672.4,E2 -5672.4} C_VEL
LIN {X 0,Y 503.824,Z 527.027,A -85,B 0,C 180,E1 -5673.299,E2 -5673.299} C_VEL
LIN {X 0,Y 504.226,Z 515.959,A -85,B 0,C 180,E1 -5673.996,E2 -5673.996} C_VEL
LIN {X 0,Y 504.434,Z 504.819,A -85,B 0,C 180,E1 -5674.545,E2 -5674.545} C_VEL
LIN {X 0,Y 504.666,Z 492.213,A -85,B 0,C 180,E1 -5674.993,E2 -5674.993} C_VEL
LIN {X 0,Y 504.912,Z 478.863,A -85,B 0,C 180,E1 -5675.291,E2 -5675.291} C_VEL
LIN {X 0,Y 505.471,Z 387.464,A -85,B 0,C 180,E1 -5676.6,E2 -5676.6} C_VEL
LIN {X 0,Y 503.338,Z 376.73,A -85,B 0,C 180,E1 -5676.836,E2 -5676.836} C_VEL
LIN {X 0,Y 503.547,Z 365.386,A -85,B 0,C 180,E1 -5679.236,E2 -5679.236} C_VEL
LIN {X 0,Y 503.048,Z 359.761,A -85,B 0,C 180,E1 -5680.464,E2 -5680.464} C_VEL
LIN {X 0,Y 502.863,Z 358.85,A -85,B 0,C 180,E1 -5680.671,E2 -5680.671} C_VEL
LIN {X 0,Y 502.837,Z 358.85,A -85,B 0,C 180,E1 -5682.922,E2 -5682.922} C_VEL
LIN {X 0,Y 502.854,Z 358.843,A -85,B 0,C 180,E1 -5685.399,E2 -5685.399} C_VEL
LIN {X 0,Y 502.846,Z 358.849,A -85,B 0,C 180,E1 -5688.12,E2 -5688.12} C_VEL
LIN {X 0,Y 502.833,Z 358.851,A -85,B 0,C 180,E1 -5690.535,E2 -5690.535} C_VEL
LIN {X 0,Y 502.801,Z 358.85,A -85,B 0,C 180,E1 -5693.04,E2 -5693.04} C_VEL
LIN {X 0,Y 502.844,Z 358.847,A -85,B 0,C 180,E1 -5695.675,E2 -5695.675} C_VEL
LIN {X 0,Y 502.845,Z 358.85,A -85,B 0,C 180,E1 -5698.372,E2 -5698.372} C_VEL
LIN {X 0,Y 502.796,Z 358.852,A -85,B 0,C 180,E1 -5701.498,E2 -5701.498} C_VEL
LIN {X 0,Y 502.808,Z 358.853,A -85,B 0,C 180,E1 -5704.444,E2 -5704.444} C_VEL
LIN {X 0,Y 502.782,Z 358.853,A -85,B 0,C 180,E1 -5707.177,E2 -5707.177} C_VEL
LIN {X 0,Y 502.787,Z 358.859,A -85,B 0,C 180,E1 -5710.014,E2 -5710.014} C_VEL
LIN {X 0,Y 502.801,Z 358.855,A -85,B 0,C 180,E1 -5712.198,E2 -5712.198} C_VEL
LIN {X 0,Y 502.799,Z 358.854,A -85,B 0,C 180,E1 -5715.467,E2 -5715.467} C_VEL
LIN {X 0,Y 502.832,Z 358.853,A -85,B 0,C 180,E1 -5717.864,E2 -5717.864} C_VEL
LIN {X 0,Y 502.806,Z 358.851,A -85,B 0,C 180,E1 -5721.024,E2 -5721.024} C_VEL
LIN {X 0,Y 502.778,Z 358.856,A -85,B 0,C 180,E1 -5724.167,E2 -5724.167} C_VEL
LIN {X 0,Y 502.828,Z 358.849,A -85,B 0,C 180,E1 -5726.992,E2 -5726.992} C_VEL
LIN {X 0,Y 502.809,Z 358.853,A -85,B 0,C 180,E1 -5730.064,E2 -5730.064} C_VEL
LIN {X 0,Y 502.829,Z 358.848,A -85,B 0,C 180,E1 -5732.533,E2 -5732.533} C_VEL
LIN {X 0,Y 502.824,Z 358.852,A -85,B 0,C 180,E1 -5735.297,E2 -5735.297} C_VEL
LIN {X 0,Y 502.803,Z 358.854,A -85,B 0,C 180,E1 -5737.827,E2 -5737.827} C_VEL
LIN {X 0,Y 502.818,Z 358.849,A -85,B 0,C 180,E1 -5740.4,E2 -5740.4} C_VEL
LIN {X 0,Y 502.829,Z 358.851,A -85,B 0,C 180,E1 -5742.931,E2 -5742.931} C_VEL
LIN {X 0,Y 502.843,Z 358.851,A -85,B 0,C 180,E1 -5745.429,E2 -5745.429} C_VEL
LIN {X 0,Y 502.886,Z 358.843,A -85,B 0,C 180,E1 -5748.717,E2 -5748.717} C_VEL
LIN {X 0,Y 502.894,Z 358.84,A -85,B 0,C 180,E1 -5751.966,E2 -5751.966} C_VEL
LIN {X 0,Y 502.931,Z 358.836,A -85,B 0,C 180,E1 -5754.386,E2 -5754.386} C_VEL
LIN {X 0,Y 503.017,Z 358.827,A -85,B 0,C 180,E1 -5757.598,E2 -5757.598} C_VEL
LIN {X 0,Y 503.017,Z 358.825,A -85,B 0,C 180,E1 -5760,E2 -5760} C_VEL
LIN {X 0,Y 503.017,Z 358.826,A -85,B 0,C 180,E1 -5762.402,E2 -5762.402} C_VEL
LIN {X 0,Y 502.94,Z 358.835,A -85,B 0,C 180,E1 -5765.613,E2 -5765.613} C_VEL
LIN {X 0,Y 502.893,Z 358.84,A -85,B 0,C 180,E1 -5768.033,E2 -5768.033} C_VEL
LIN {X 0,Y 502.886,Z 358.843,A -85,B 0,C 180,E1 -5771.283,E2 -5771.283} C_VEL
LIN {X 0,Y 502.842,Z 358.852,A -85,B 0,C 180,E1 -5774.571,E2 -5774.571} C_VEL
LIN {X 0,Y 502.853,Z 358.845,A -85,B 0,C 180,E1 -5777.907,E2 -5777.907} C_VEL
LIN {X 0,Y 502.822,Z 358.854,A -85,B 0,C 180,E1 -5780.537,E2 -5780.537} C_VEL
LIN {X 0,Y 502.798,Z 358.854,A -85,B 0,C 180,E1 -5783.04,E2 -5783.04} C_VEL
LIN {X 0,Y 502.834,Z 358.847,A -85,B 0,C 180,E1 -5785.676,E2 -5785.676} C_VEL
LIN {X 0,Y 502.833,Z 358.853,A -85,B 0,C 180,E1 -5788.373,E2 -5788.373} C_VEL
LIN {X 0,Y 502.789,Z 358.852,A -85,B 0,C 180,E1 -5791.5,E2 -5791.5} C_VEL
LIN {X 0,Y 502.8,Z 358.856,A -85,B 0,C 180,E1 -5794.445,E2 -5794.445} C_VEL
LIN {X 0,Y 502.775,Z 358.854,A -85,B 0,C 180,E1 -5797.179,E2 -5797.179} C_VEL
LIN {X 0,Y 502.816,Z 358.854,A -85,B 0,C 180,E1 -5800.013,E2 -5800.013} C_VEL
LIN {X 0,Y 502.818,Z 358.855,A -85,B 0,C 180,E1 -5802.203,E2 -5802.203} C_VEL
LIN {X 0,Y 502.796,Z 358.852,A -85,B 0,C 180,E1 -5805.469,E2 -5805.469} C_VEL
LIN {X 0,Y 502.817,Z 358.848,A -85,B 0,C 180,E1 -5808.935,E2 -5808.935} C_VEL
LIN {X 0,Y 502.792,Z 358.858,A -85,B 0,C 180,E1 -5812.047,E2 -5812.047} C_VEL
LIN {X 0,Y 502.808,Z 358.849,A -85,B 0,C 180,E1 -5815.036,E2 -5815.036} C_VEL
LIN {X 0,Y 502.787,Z 358.86,A -85,B 0,C 180,E1 -5817.917,E2 -5817.917} C_VEL
LIN {X 0,Y 502.839,Z 358.847,A -85,B 0,C 180,E1 -5820.714,E2 -5820.714} C_VEL
LIN {X 0,Y 502.862,Z 358.848,A -85,B 0,C 180,E1 -5823.44,E2 -5823.44} C_VEL
LIN {X 0,Y 502.903,Z 358.893,A -85,B 0,C 180,E1 -5824.387,E2 -5824.387} C_VEL
LIN {X 0,Y 504.778,Z 369.47,A -85,B 0,C 180,E1 -5826.187,E2 -5826.187} C_VEL
LIN {X 0,Y 504.212,Z 387.52,A -85,B 0,C 180,E1 -5829.049,E2 -5829.049} C_VEL
LIN {X 0,Y 503.616,Z 408.494,A -85,B 0,C 180,E1 -5832.331,E2 -5832.331} C_VEL
LIN {X 0,Y 503.279,Z 420.566,A -85,B 0,C 180,E1 -5834.192,E2 -5834.192} C_VEL
LIN {X 0,Y 505.4,Z 435.215,A -85,B 0,C 180,E1 -5834.47,E2 -5834.47} C_VEL
LIN {X 0,Y 504.856,Z 528.967,A -85,B 0,C 180,E1 -5835.823,E2 -5835.823} C_VEL
LIN {X 0,Y 504.569,Z 542.295,A -85,B 0,C 180,E1 -5836.175,E2 -5836.175} C_VEL
LIN {X 0,Y 504.216,Z 555.624,A -85,B 0,C 180,E1 -5836.704,E2 -5836.704} C_VEL
LIN {X 0,Y 503.852,Z 568.17,A -85,B 0,C 180,E1 -5837.397,E2 -5837.397} C_VEL
LIN {X 0,Y 503.491,Z 579.745,A -85,B 0,C 180,E1 -5838.221,E2 -5838.221} C_VEL
LIN {X 0,Y 503.166,Z 589.975,A -85,B 0,C 180,E1 -5839.131,E2 -5839.131} C_VEL
LIN {X 0,Y 502.847,Z 599.18,A -85,B 0,C 180,E1 -5840.142,E2 -5840.142} C_VEL
LIN {X 0,Y 502.552,Z 608.152,A -85,B 0,C 180,E1 -5841.354,E2 -5841.354} C_VEL
LIN {X 0,Y 502.349,Z 615.376,A -85,B 0,C 180,E1 -5842.565,E2 -5842.565} C_VEL
LIN {X 0,Y 502.235,Z 620.253,A -85,B 0,C 180,E1 -5843.573,E2 -5843.573} C_VEL
LIN {X 0,Y 502.175,Z 624.995,A -85,B 0,C 180,E1 -5844.781,E2 -5844.781} C_VEL
LIN {X 0,Y 502.164,Z 628.619,A -85,B 0,C 180,E1 -5845.987,E2 -5845.987} C_VEL
LIN {X 0,Y 502.122,Z 630.487,A -85,B 0,C 180,E1 -5846.791,E2 -5846.791} C_VEL
LIN {X 0,Y 502.12,Z 631.889,A -85,B 0,C 180,E1 -5847.594,E2 -5847.594} C_VEL
LIN {X 0,Y 501.99,Z 633.492,A -85,B 0,C 180,E1 -5849.198,E2 -5849.198} C_VEL
LIN {X 0,Y 501.983,Z 633.707,A -85,B 0,C 180,E1 -5850,E2 -5850} C_VEL
LIN {X 0,Y 502.036,Z 632.88,A -85,B 0,C 180,E1 -5851.604,E2 -5851.604} C_VEL
LIN {X 0,Y 502.12,Z 631.883,A -85,B 0,C 180,E1 -5852.406,E2 -5852.406} C_VEL
LIN {X 0,Y 502.122,Z 630.479,A -85,B 0,C 180,E1 -5853.209,E2 -5853.209} C_VEL
LIN {X 0,Y 502.104,Z 627.526,A -85,B 0,C 180,E1 -5854.415,E2 -5854.415} C_VEL
LIN {X 0,Y 502.211,Z 623.536,A -85,B 0,C 180,E1 -5855.622,E2 -5855.622} C_VEL
LIN {X 0,Y 502.333,Z 617.499,A -85,B 0,C 180,E1 -5857.011,E2 -5857.011} C_VEL
LIN {X 0,Y 502.482,Z 610.69,A -85,B 0,C 180,E1 -5858.242,E2 -5858.242} C_VEL
LIN {X 0,Y 502.719,Z 602.373,A -85,B 0,C 180,E1 -5859.454,E2 -5859.454} C_VEL
LIN {X 0,Y 502.994,Z 593.852,A -85,B 0,C 180,E1 -5860.465,E2 -5860.465} C_VEL
LIN {X 0,Y 503.406,Z 583.329,A -85,B 0,C 180,E1 -5861.475,E2 -5861.475} C_VEL
LIN {X 0,Y 503.679,Z 572.116,A -85,B 0,C 180,E1 -5862.343,E2 -5862.343} C_VEL
LIN {X 0,Y 504.058,Z 561.514,A -85,B 0,C 180,E1 -5862.992,E2 -5862.992} C_VEL
LIN {X 0,Y 504.362,Z 549.808,A -85,B 0,C 180,E1 -5863.548,E2 -5863.548} C_VEL
LIN {X 0,Y 504.697,Z 536.331,A -85,B 0,C 180,E1 -5864.001,E2 -5864.001} C_VEL
LIN {X 0,Y 504.92,Z 522.984,A -85,B 0,C 180,E1 -5864.278,E2 -5864.278} C_VEL
LIN {X 0,Y 505.359,Z 434.109,A -85,B 0,C 180,E1 -5865.546,E2 -5865.546} C_VEL
LIN {X 0,Y 503.262,Z 420.314,A -85,B 0,C 180,E1 -5865.827,E2 -5865.827} C_VEL
LIN {X 0,Y 503.792,Z 400.366,A -85,B 0,C 180,E1 -5868.925,E2 -5868.925} C_VEL
LIN {X 0,Y 504.396,Z 381.608,A -85,B 0,C 180,E1 -5871.883,E2 -5871.883} C_VEL
LIN {X 0,Y 504.836,Z 369.573,A -85,B 0,C 180,E1 -5873.81,E2 -5873.81} C_VEL
LIN {X 0,Y 502.895,Z 358.845,A -85,B 0,C 180,E1 -5875.7,E2 -5875.7} C_VEL
LIN {X 0,Y 502.842,Z 358.85,A -85,B 0,C 180,E1 -5878.372,E2 -5878.372} C_VEL
LIN {X 0,Y 502.797,Z 358.851,A -85,B 0,C 180,E1 -5881.499,E2 -5881.499} C_VEL
LIN {X 0,Y 502.805,Z 358.853,A -85,B 0,C 180,E1 -5884.444,E2 -5884.444} C_VEL
LIN {X 0,Y 502.779,Z 358.854,A -85,B 0,C 180,E1 -5887.178,E2 -5887.178} C_VEL
LIN {X 0,Y 502.785,Z 358.857,A -85,B 0,C 180,E1 -5890.014,E2 -5890.014} C_VEL
LIN {X 0,Y 502.799,Z 358.852,A -85,B 0,C 180,E1 -5892.198,E2 -5892.198} C_VEL
LIN {X 0,Y 502.796,Z 358.853,A -85,B 0,C 180,E1 -5895.467,E2 -5895.467} C_VEL
LIN {X 0,Y 502.83,Z 358.851,A -85,B 0,C 180,E1 -5897.864,E2 -5897.864} C_VEL
LIN {X 0,Y 502.804,Z 358.849,A -85,B 0,C 180,E1 -5901.024,E2 -5901.024} C_VEL
LIN {X 0,Y 502.78,Z 358.853,A -85,B 0,C 180,E1 -5904.166,E2 -5904.166} C_VEL
LIN {X 0,Y 502.826,Z 358.848,A -85,B 0,C 180,E1 -5906.993,E2 -5906.993} C_VEL
LIN {X 0,Y 502.823,Z 358.848,A -85,B 0,C 180,E1 -5910.061,E2 -5910.061} C_VEL
LIN {X 0,Y 502.828,Z 358.846,A -85,B 0,C 180,E1 -5912.533,E2 -5912.533} C_VEL
LIN {X 0,Y 502.823,Z 358.844,A -85,B 0,C 180,E1 -5915.297,E2 -5915.297} C_VEL
LIN {X 0,Y 502.802,Z 358.851,A -85,B 0,C 180,E1 -5917.828,E2 -5917.828} C_VEL
LIN {X 0,Y 502.817,Z 358.846,A -85,B 0,C 180,E1 -5920.4,E2 -5920.4} C_VEL
LIN {X 0,Y 502.828,Z 358.851,A -85,B 0,C 180,E1 -5922.932,E2 -5922.932} C_VEL
LIN {X 0,Y 502.836,Z 358.849,A -85,B 0,C 180,E1 -5925.429,E2 -5925.429} C_VEL
LIN {X 0,Y 502.888,Z 358.842,A -85,B 0,C 180,E1 -5928.717,E2 -5928.717} C_VEL
LIN {X 0,Y 502.893,Z 358.838,A -85,B 0,C 180,E1 -5931.967,E2 -5931.967} C_VEL
LIN {X 0,Y 502.931,Z 358.832,A -85,B 0,C 180,E1 -5934.387,E2 -5934.387} C_VEL
LIN {X 0,Y 503.017,Z 358.822,A -85,B 0,C 180,E1 -5937.598,E2 -5937.598} C_VEL
LIN {X 0,Y 503.017,Z 358.822,A -85,B 0,C 180,E1 -5940,E2 -5940} C_VEL
LIN {X 0,Y 503.017,Z 358.826,A -85,B 0,C 180,E1 -5942.402,E2 -5942.402} C_VEL
LIN {X 0,Y 502.931,Z 358.833,A -85,B 0,C 180,E1 -5945.614,E2 -5945.614} C_VEL
LIN {X 0,Y 502.894,Z 358.837,A -85,B 0,C 180,E1 -5948.034,E2 -5948.034} C_VEL
LIN {X 0,Y 502.873,Z 358.841,A -85,B 0,C 180,E1 -5951.284,E2 -5951.284} C_VEL
LIN {X 0,Y 502.843,Z 358.852,A -85,B 0,C 180,E1 -5954.571,E2 -5954.571} C_VEL
LIN {X 0,Y 502.854,Z 358.843,A -85,B 0,C 180,E1 -5957.908,E2 -5957.908} C_VEL
LIN {X 0,Y 502.821,Z 358.852,A -85,B 0,C 180,E1 -5960.537,E2 -5960.537} C_VEL
LIN {X 0,Y 502.789,Z 358.852,A -85,B 0,C 180,E1 -5963.041,E2 -5963.041} C_VEL
LIN {X 0,Y 502.835,Z 358.842,A -85,B 0,C 180,E1 -5965.676,E2 -5965.676} C_VEL
LIN {X 0,Y 502.834,Z 358.851,A -85,B 0,C 180,E1 -5968.373,E2 -5968.373} C_VEL
LIN {X 0,Y 502.791,Z 358.85,A -85,B 0,C 180,E1 -5971.5,E2 -5971.5} C_VEL
LIN {X 0,Y 502.801,Z 358.855,A -85,B 0,C 180,E1 -5974.446,E2 -5974.446} C_VEL
LIN {X 0,Y 502.777,Z 358.853,A -85,B 0,C 180,E1 -5977.179,E2 -5977.179} C_VEL
LIN {X 0,Y 502.819,Z 358.856,A -85,B 0,C 180,E1 -5980.013,E2 -5980.013} C_VEL
LIN {X 0,Y 502.82,Z 358.851,A -85,B 0,C 180,E1 -5982.203,E2 -5982.203} C_VEL
LIN {X 0,Y 502.799,Z 358.855,A -85,B 0,C 180,E1 -5985.469,E2 -5985.469} C_VEL
LIN {X 0,Y 502.826,Z 358.849,A -85,B 0,C 180,E1 -5989.005,E2 -5989.005} C_VEL
LIN {X 0,Y 502.797,Z 358.857,A -85,B 0,C 180,E1 -5992.047,E2 -5992.047} C_VEL
LIN {X 0,Y 502.811,Z 358.851,A -85,B 0,C 180,E1 -5995.036,E2 -5995.036} C_VEL
LIN {X 0,Y 502.809,Z 358.85,A -85,B 0,C 180,E1 -5997.24,E2 -5997.24} C_VEL
LIN {X 0,Y 502.108,Z 358.943,A -85,B 0,C 180,E1 -5997.909,E2 -5997.909} C_VEL
LIN {X 0,Y 499.244,Z 359.297,A -85,B 0,C 180,E1 -5998.995,E2 -5998.995} C_VEL
LIN {X 0,Y 496.859,Z 359.597,A -85,B 0,C 180,E1 -5999.87,E2 -5999.87} C_VEL
LIN {X 0,Y 495.86,Z 359.719,A -85,B 0,C 180,E1 -6000.545,E2 -6000.545} C_VEL
LIN {X 0,Y 495.791,Z 359.727,A -85,B 0,C 180,E1 -6000.774,E2 -6000.774} C_VEL
LIN {X 0,Y 495.842,Z 359.832,A -85,B 0,C 180,E1 -6001.236,E2 -6001.236} C_VEL
LIN {X 0,Y 496.654,Z 364.911,A -85,B 0,C 180,E1 -6002.392,E2 -6002.392} C_VEL
LIN {X 0,Y 496.34,Z 377.12,A -85,B 0,C 180,E1 -6005.018,E2 -6005.018} C_VEL
LIN {X 0,Y 498.689,Z 389.781,A -85,B 0,C 180,E1 -6005.3,E2 -6005.3} C_VEL
LIN {X 0,Y 498.044,Z 483.351,A -85,B 0,C 180,E1 -6006.672,E2 -6006.672} C_VEL
LIN {X 0,Y 497.826,Z 496.266,A -85,B 0,C 180,E1 -6007.019,E2 -6007.019} C_VEL
LIN {X 0,Y 497.539,Z 508.917,A -85,B 0,C 180,E1 -6007.526,E2 -6007.526} C_VEL
LIN {X 0,Y 497.264,Z 519.816,A -85,B 0,C 180,E1 -6008.114,E2 -6008.114} C_VEL
LIN {X 0,Y 496.893,Z 531.099,A -85,B 0,C 180,E1 -6008.895,E2 -6008.895} C_VEL
LIN {X 0,Y 496.491,Z 541.686,A -85,B 0,C 180,E1 -6009.816,E2 -6009.816} C_VEL
LIN {X 0,Y 496.148,Z 550.625,A -85,B 0,C 180,E1 -6010.772,E2 -6010.772} C_VEL
LIN {X 0,Y 495.809,Z 558.782,A -85,B 0,C 180,E1 -6011.83,E2 -6011.83} C_VEL
LIN {X 0,Y 495.55,Z 566.674,A -85,B 0,C 180,E1 -6013.098,E2 -6013.098} C_VEL
LIN {X 0,Y 495.338,Z 572.934,A -85,B 0,C 180,E1 -6014.361,E2 -6014.361} C_VEL
LIN {X 0,Y 495.187,Z 577.855,A -85,B 0,C 180,E1 -6015.619,E2 -6015.619} C_VEL
LIN {X 0,Y 495.09,Z 581.6,A -85,B 0,C 180,E1 -6016.872,E2 -6016.872} C_VEL
LIN {X 0,Y 495.046,Z 584.773,A -85,B 0,C 180,E1 -6018.401,E2 -6018.401} C_VEL
LIN {X 0,Y 494.996,Z 585.988,A -85,B 0,C 180,E1 -6019.364,E2 -6019.364} C_VEL
LIN {X 0,Y 494.96,Z 586.844,A -85,B 0,C 180,E1 -6021.014,E2 -6021.014} C_VEL
LIN {X 0,Y 495,Z 586.641,A -85,B 0,C 180,E1 -6021.838,E2 -6021.838} C_VEL
LIN {X 0,Y 495.079,Z 585.054,A -85,B 0,C 180,E1 -6023.479,E2 -6023.479} C_VEL
LIN {X 0,Y 495.114,Z 583.675,A -85,B 0,C 180,E1 -6024.298,E2 -6024.298} C_VEL
LIN {X 0,Y 495.113,Z 580.787,A -85,B 0,C 180,E1 -6025.522,E2 -6025.522} C_VEL
LIN {X 0,Y 495.254,Z 576.872,A -85,B 0,C 180,E1 -6026.746,E2 -6026.746} C_VEL
LIN {X 0,Y 495.298,Z 571.859,A -85,B 0,C 180,E1 -6027.967,E2 -6027.967} C_VEL
LIN {X 0,Y 495.599,Z 565.533,A -85,B 0,C 180,E1 -6029.187,E2 -6029.187} C_VEL
LIN {X 0,Y 495.836,Z 557.684,A -85,B 0,C 180,E1 -6030.406,E2 -6030.406} C_VEL
LIN {X 0,Y 496.243,Z 547.935,A -85,B 0,C 180,E1 -6031.623,E2 -6031.623} C_VEL
LIN {X 0,Y 496.533,Z 537.762,A -85,B 0,C 180,E1 -6032.637,E2 -6032.637} C_VEL
LIN {X 0,Y 496.937,Z 526.305,A -85,B 0,C 180,E1 -6033.547,E2 -6033.547} C_VEL
LIN {X 0,Y 497.384,Z 514.952,A -85,B 0,C 180,E1 -6034.254,E2 -6034.254} C_VEL
LIN {X 0,Y 497.56,Z 503.315,A -85,B 0,C 180,E1 -6034.811,E2 -6034.811} C_VEL
LIN {X 0,Y 497.862,Z 489.823,A -85,B 0,C 180,E1 -6035.265,E2 -6035.265} C_VEL
LIN {X 0,Y 498.062,Z 477.706,A -85,B 0,C 180,E1 -6035.516,E2 -6035.516} C_VEL
LIN {X 0,Y 498.529,Z 387.422,A -85,B 0,C 180,E1 -6036.826,E2 -6036.826} C_VEL
LIN {X 0,Y 496.337,Z 377.036,A -85,B 0,C 180,E1 -6037.062,E2 -6037.062} C_VEL
LIN {X 0,Y 496.574,Z 366.247,A -85,B 0,C 180,E1 -6039.367,E2 -6039.367} C_VEL
LIN {X 0,Y 495.985,Z 360.608,A -85,B 0,C 180,E1 -6040.615,E2 -6040.615} C_VEL
LIN {X 0,Y 495.829,Z 359.727,A -85,B 0,C 180,E1 -6040.825,E2 -6040.825} C_VEL
LIN {X 0,Y 495.799,Z 359.727,A -85,B 0,C 180,E1 -6043.944,E2 -6043.944} C_VEL
LIN {X 0,Y 495.783,Z 359.731,A -85,B 0,C 180,E1 -6046.469,E2 -6046.469} C_VEL
LIN {X 0,Y 495.788,Z 359.724,A -85,B 0,C 180,E1 -6049.028,E2 -6049.028} C_VEL
LIN {X 0,Y 495.748,Z 359.729,A -85,B 0,C 180,E1 -6051.628,E2 -6051.628} C_VEL
LIN {X 0,Y 495.783,Z 359.725,A -85,B 0,C 180,E1 -6054.873,E2 -6054.873} C_VEL
LIN {X 0,Y 495.817,Z 359.72,A -85,B 0,C 180,E1 -6056.973,E2 -6056.973} C_VEL
LIN {X 0,Y 495.779,Z 359.732,A -85,B 0,C 180,E1 -6060.149,E2 -6060.149} C_VEL
LIN {X 0,Y 495.795,Z 359.724,A -85,B 0,C 180,E1 -6063.244,E2 -6063.244} C_VEL
LIN {X 0,Y 495.73,Z 359.738,A -85,B 0,C 180,E1 -6066.089,E2 -6066.089} C_VEL
LIN {X 0,Y 495.764,Z 359.728,A -85,B 0,C 180,E1 -6068.767,E2 -6068.767} C_VEL
LIN {X 0,Y 495.755,Z 359.733,A -85,B 0,C 180,E1 -6071.78,E2 -6071.78} C_VEL
LIN {X 0,Y 495.747,Z 359.731,A -85,B 0,C 180,E1 -6075.138,E2 -6075.138} C_VEL
LIN {X 0,Y 495.779,Z 359.729,A -85,B 0,C 180,E1 -6078.221,E2 -6078.221} C_VEL
LIN {X 0,Y 495.765,Z 359.73,A -85,B 0,C 180,E1 -6081.23,E2 -6081.23} C_VEL
LIN {X 0,Y 495.75,Z 359.73,A -85,B 0,C 180,E1 -6084.462,E2 -6084.462} C_VEL
LIN {X 0,Y 495.764,Z 359.731,A -85,B 0,C 180,E1 -6087.405,E2 -6087.405} C_VEL
LIN {X 0,Y 495.76,Z 359.729,A -85,B 0,C 180,E1 -6090.253,E2 -6090.253} C_VEL
LIN {X 0,Y 495.827,Z 359.723,A -85,B 0,C 180,E1 -6093.247,E2 -6093.247} C_VEL
LIN {X 0,Y 495.753,Z 359.735,A -85,B 0,C 180,E1 -6095.725,E2 -6095.725} C_VEL
LIN {X 0,Y 495.753,Z 359.73,A -85,B 0,C 180,E1 -6098.371,E2 -6098.371} C_VEL
LIN {X 0,Y 495.777,Z 359.73,A -85,B 0,C 180,E1 -6100.971,E2 -6100.971} C_VEL
LIN {X 0,Y 495.773,Z 359.731,A -85,B 0,C 180,E1 -6103.529,E2 -6103.529} C_VEL
LIN {X 0,Y 495.793,Z 359.725,A -85,B 0,C 180,E1 -6106.055,E2 -6106.055} C_VEL
LIN {X 0,Y 495.867,Z 359.717,A -85,B 0,C 180,E1 -6108.555,E2 -6108.555} C_VEL
LIN {X 0,Y 495.865,Z 359.717,A -85,B 0,C 180,E1 -6111.852,E2 -6111.852} C_VEL
LIN {X 0,Y 495.889,Z 359.713,A -85,B 0,C 180,E1 -6114.306,E2 -6114.306} C_VEL
LIN {X 0,Y 495.986,Z 359.703,A -85,B 0,C 180,E1 -6117.563,E2 -6117.563} C_VEL
LIN {X 0,Y 495.988,Z 359.7,A -85,B 0,C 180,E1 -6120,E2 -6120} C_VEL
LIN {X 0,Y 495.986,Z 359.703,A -85,B 0,C 180,E1 -6122.436,E2 -6122.436} C_VEL
LIN {X 0,Y 495.896,Z 359.712,A -85,B 0,C 180,E1 -6125.693,E2 -6125.693} C_VEL
LIN {X 0,Y 495.865,Z 359.716,A -85,B 0,C 180,E1 -6128.148,E2 -6128.148} C_VEL
LIN {X 0,Y 495.866,Z 359.717,A -85,B 0,C 180,E1 -6131.445,E2 -6131.445} C_VEL
LIN {X 0,Y 495.785,Z 359.729,A -85,B 0,C 180,E1 -6134.783,E2 -6134.783} C_VEL
LIN {X 0,Y 495.78,Z 359.727,A -85,B 0,C 180,E1 -6137.319,E2 -6137.319} C_VEL
LIN {X 0,Y 495.769,Z 359.728,A -85,B 0,C 180,E1 -6139.89,E2 -6139.89} C_VEL
LIN {X 0,Y 495.756,Z 359.732,A -85,B 0,C 180,E1 -6142.863,E2 -6142.863} C_VEL
LIN {X 0,Y 495.792,Z 359.727,A -85,B 0,C 180,E1 -6146.068,E2 -6146.068} C_VEL
LIN {X 0,Y 495.764,Z 359.73,A -85,B 0,C 180,E1 -6148.815,E2 -6148.815} C_VEL
LIN {X 0,Y 495.751,Z 359.73,A -85,B 0,C 180,E1 -6151.727,E2 -6151.727} C_VEL
LIN {X 0,Y 495.77,Z 359.729,A -85,B 0,C 180,E1 -6154.696,E2 -6154.696} C_VEL
LIN {X 0,Y 495.726,Z 359.733,A -85,B 0,C 180,E1 -6157.562,E2 -6157.562} C_VEL
LIN {X 0,Y 495.774,Z 359.728,A -85,B 0,C 180,E1 -6160.699,E2 -6160.699} C_VEL
LIN {X 0,Y 495.73,Z 359.733,A -85,B 0,C 180,E1 -6163.696,E2 -6163.696} C_VEL
LIN {X 0,Y 495.724,Z 359.736,A -85,B 0,C 180,E1 -6166.306,E2 -6166.306} C_VEL
LIN {X 0,Y 495.763,Z 359.727,A -85,B 0,C 180,E1 -6169.301,E2 -6169.301} C_VEL
LIN {X 0,Y 495.729,Z 359.734,A -85,B 0,C 180,E1 -6172.439,E2 -6172.439} C_VEL
LIN {X 0,Y 495.784,Z 359.726,A -85,B 0,C 180,E1 -6175.458,E2 -6175.458} C_VEL
LIN {X 0,Y 495.759,Z 359.729,A -85,B 0,C 180,E1 -6178.365,E2 -6178.365} C_VEL
LIN {X 0,Y 495.79,Z 359.728,A -85,B 0,C 180,E1 -6181.507,E2 -6181.507} C_VEL
LIN {X 0,Y 495.839,Z 359.823,A -85,B 0,C 180,E1 -6184.218,E2 -6184.218} C_VEL
LIN {X 0,Y 497.813,Z 370.584,A -85,B 0,C 180,E1 -6186.076,E2 -6186.076} C_VEL
LIN {X 0,Y 497.267,Z 387.995,A -85,B 0,C 180,E1 -6188.875,E2 -6188.875} C_VEL
LIN {X 0,Y 496.606,Z 409.51,A -85,B 0,C 180,E1 -6192.286,E2 -6192.286} C_VEL
LIN {X 0,Y 496.276,Z 420.238,A -85,B 0,C 180,E1 -6193.964,E2 -6193.964} C_VEL
LIN {X 0,Y 498.556,Z 436.2,A -85,B 0,C 180,E1 -6194.271,E2 -6194.271} C_VEL
LIN {X 0,Y 497.972,Z 528.616,A -85,B 0,C 180,E1 -6195.623,E2 -6195.623} C_VEL
LIN {X 0,Y 497.669,Z 541.95,A -85,B 0,C 180,E1 -6195.979,E2 -6195.979} C_VEL
LIN {X 0,Y 497.284,Z 555.283,A -85,B 0,C 180,E1 -6196.515,E2 -6196.515} C_VEL
LIN {X 0,Y 496.872,Z 567.835,A -85,B 0,C 180,E1 -6197.217,E2 -6197.217} C_VEL
LIN {X 0,Y 496.488,Z 579.407,A -85,B 0,C 180,E1 -6198.052,E2 -6198.052} C_VEL
LIN {X 0,Y 496.17,Z 589.64,A -85,B 0,C 180,E1 -6198.976,E2 -6198.976} C_VEL
LIN {X 0,Y 495.791,Z 598.844,A -85,B 0,C 180,E1 -6200,E2 -6200} C_VEL
LIN {X 0,Y 495.481,Z 607.816,A -85,B 0,C 180,E1 -6201.23,E2 -6201.23} C_VEL
LIN {X 0,Y 495.28,Z 615.042,A -85,B 0,C 180,E1 -6202.458,E2 -6202.458} C_VEL
LIN {X 0,Y 495.124,Z 621.101,A -85,B 0,C 180,E1 -6203.758,E2 -6203.758} C_VEL
LIN {X 0,Y 495.037,Z 625.978,A -85,B 0,C 180,E1 -6205.114,E2 -6205.114} C_VEL
LIN {X 0,Y 495.055,Z 628.286,A -85,B 0,C 180,E1 -6205.93,E2 -6205.93} C_VEL
LIN {X 0,Y 495.045,Z 630.155,A -85,B 0,C 180,E1 -6206.745,E2 -6206.745} C_VEL
LIN {X 0,Y 495.024,Z 631.556,A -85,B 0,C 180,E1 -6207.559,E2 -6207.559} C_VEL
LIN {X 0,Y 494.91,Z 633.159,A -85,B 0,C 180,E1 -6209.186,E2 -6209.186} C_VEL
LIN {X 0,Y 494.901,Z 633.375,A -85,B 0,C 180,E1 -6210,E2 -6210} C_VEL
LIN {X 0,Y 494.963,Z 632.547,A -85,B 0,C 180,E1 -6211.627,E2 -6211.627} C_VEL
LIN {X 0,Y 495.024,Z 631.547,A -85,B 0,C 180,E1 -6212.441,E2 -6212.441} C_VEL
LIN {X 0,Y 495.045,Z 630.144,A -85,B 0,C 180,E1 -6213.255,E2 -6213.255} C_VEL
LIN {X 0,Y 495.009,Z 627.189,A -85,B 0,C 180,E1 -6214.479,E2 -6214.479} C_VEL
LIN {X 0,Y 495.127,Z 623.197,A -85,B 0,C 180,E1 -6215.702,E2 -6215.702} C_VEL
LIN {X 0,Y 495.256,Z 617.057,A -85,B 0,C 180,E1 -6217.133,E2 -6217.133} C_VEL
LIN {X 0,Y 495.428,Z 610.349,A -85,B 0,C 180,E1 -6218.36,E2 -6218.36} C_VEL
LIN {X 0,Y 495.681,Z 602.03,A -85,B 0,C 180,E1 -6219.59,E2 -6219.59} C_VEL
LIN {X 0,Y 495.985,Z 593.507,A -85,B 0,C 180,E1 -6220.615,E2 -6220.615} C_VEL
LIN {X 0,Y 496.425,Z 582.983,A -85,B 0,C 180,E1 -6221.638,E2 -6221.638} C_VEL
LIN {X 0,Y 496.699,Z 572.087,A -85,B 0,C 180,E1 -6222.496,E2 -6222.496} C_VEL
LIN {X 0,Y 497.101,Z 561.162,A -85,B 0,C 180,E1 -6223.178,E2 -6223.178} C_VEL
LIN {X 0,Y 497.439,Z 549.454,A -85,B 0,C 180,E1 -6223.741,E2 -6223.741} C_VEL
LIN {X 0,Y 497.783,Z 536.888,A -85,B 0,C 180,E1 -6224.174,E2 -6224.174} C_VEL
LIN {X 0,Y 498.039,Z 524.148,A -85,B 0,C 180,E1 -6224.453,E2 -6224.453} C_VEL
LIN {X 0,Y 498.485,Z 434.84,A -85,B 0,C 180,E1 -6225.75,E2 -6225.75} C_VEL
LIN {X 0,Y 496.262,Z 420.064,A -85,B 0,C 180,E1 -6226.045,E2 -6226.045} C_VEL
LIN {X 0,Y 496.857,Z 400.088,A -85,B 0,C 180,E1 -6229.2,E2 -6229.2} C_VEL
LIN {X 0,Y 497.462,Z 382.721,A -85,B 0,C 180,E1 -6231.986,E2 -6231.986} C_VEL
LIN {X 0,Y 497.896,Z 370.72,A -85,B 0,C 180,E1 -6233.942,E2 -6233.942} C_VEL
LIN {X 0,Y 495.854,Z 359.723,A -85,B 0,C 180,E1 -6235.894,E2 -6235.894} C_VEL
LIN {X 0,Y 495.78,Z 359.726,A -85,B 0,C 180,E1 -6238.814,E2 -6238.814} C_VEL
LIN {X 0,Y 495.758,Z 359.73,A -85,B 0,C 180,E1 -6241.726,E2 -6241.726} C_VEL
LIN {X 0,Y 495.775,Z 359.727,A -85,B 0,C 180,E1 -6244.695,E2 -6244.695} C_VEL
LIN {X 0,Y 495.729,Z 359.735,A -85,B 0,C 180,E1 -6247.561,E2 -6247.561} C_VEL
LIN {X 0,Y 495.763,Z 359.726,A -85,B 0,C 180,E1 -6250.699,E2 -6250.699} C_VEL
LIN {X 0,Y 495.729,Z 359.734,A -85,B 0,C 180,E1 -6254,E2 -6254} C_VEL
LIN {X 0,Y 495.758,Z 359.727,A -85,B 0,C 180,E1 -6257.12,E2 -6257.12} C_VEL
LIN {X 0,Y 495.777,Z 359.724,A -85,B 0,C 180,E1 -6260.364,E2 -6260.364} C_VEL
LIN {X 0,Y 495.728,Z 359.736,A -85,B 0,C 180,E1 -6263.456,E2 -6263.456} C_VEL
LIN {X 0,Y 495.754,Z 359.727,A -85,B 0,C 180,E1 -6266.435,E2 -6266.435} C_VEL
LIN {X 0,Y 495.75,Z 359.734,A -85,B 0,C 180,E1 -6269.313,E2 -6269.313} C_VEL
LIN {X 0,Y 495.775,Z 359.725,A -85,B 0,C 180,E1 -6272.108,E2 -6272.108} C_VEL
LIN {X 0,Y 495.782,Z 359.719,A -85,B 0,C 180,E1 -6274.832,E2 -6274.832} C_VEL
LIN {X 0,Y 495.752,Z 359.734,A -85,B 0,C 180,E1 -6277.495,E2 -6277.495} C_VEL
LIN {X 0,Y 495.769,Z 359.724,A -85,B 0,C 180,E1 -6280.11,E2 -6280.11} C_VEL
LIN {X 0,Y 495.779,Z 359.726,A -85,B 0,C 180,E1 -6282.681,E2 -6282.681} C_VEL
LIN {X 0,Y 495.781,Z 359.729,A -85,B 0,C 180,E1 -6285.217,E2 -6285.217} C_VEL
LIN {X 0,Y 495.868,Z 359.715,A -85,B 0,C 180,E1 -6288.555,E2 -6288.555} C_VEL
LIN {X 0,Y 495.865,Z 359.714,A -85,B 0,C 180,E1 -6291.852,E2 -6291.852} C_VEL
LIN {X 0,Y 495.888,Z 359.708,A -85,B 0,C 180,E1 -6294.307,E2 -6294.307} C_VEL
LIN {X 0,Y 495.986,Z 359.698,A -85,B 0,C 180,E1 -6297.564,E2 -6297.564} C_VEL
LIN {X 0,Y 495.988,Z 359.697,A -85,B 0,C 180,E1 -6300,E2 -6300} C_VEL
LIN {X 0,Y 495.986,Z 359.702,A -85,B 0,C 180,E1 -6302.437,E2 -6302.437} C_VEL
LIN {X 0,Y 495.889,Z 359.711,A -85,B 0,C 180,E1 -6305.694,E2 -6305.694} C_VEL
LIN {X 0,Y 495.865,Z 359.713,A -85,B 0,C 180,E1 -6308.148,E2 -6308.148} C_VEL
LIN {X 0,Y 495.846,Z 359.715,A -85,B 0,C 180,E1 -6311.446,E2 -6311.446} C_VEL
LIN {X 0,Y 495.786,Z 359.729,A -85,B 0,C 180,E1 -6314.783,E2 -6314.783} C_VEL
LIN {X 0,Y 495.78,Z 359.723,A -85,B 0,C 180,E1 -6317.319,E2 -6317.319} C_VEL
LIN {X 0,Y 495.77,Z 359.727,A -85,B 0,C 180,E1 -6319.891,E2 -6319.891} C_VEL
LIN {X 0,Y 495.751,Z 359.73,A -85,B 0,C 180,E1 -6322.861,E2 -6322.861} C_VEL
LIN {X 0,Y 495.793,Z 359.722,A -85,B 0,C 180,E1 -6326.068,E2 -6326.068} C_VEL
LIN {X 0,Y 495.766,Z 359.728,A -85,B 0,C 180,E1 -6328.816,E2 -6328.816} C_VEL
LIN {X 0,Y 495.753,Z 359.728,A -85,B 0,C 180,E1 -6331.727,E2 -6331.727} C_VEL
LIN {X 0,Y 495.771,Z 359.728,A -85,B 0,C 180,E1 -6334.696,E2 -6334.696} C_VEL
LIN {X 0,Y 495.728,Z 359.733,A -85,B 0,C 180,E1 -6337.562,E2 -6337.562} C_VEL
LIN {X 0,Y 495.777,Z 359.727,A -85,B 0,C 180,E1 -6340.699,E2 -6340.699} C_VEL
LIN {X 0,Y 495.732,Z 359.735,A -85,B 0,C 180,E1 -6343.696,E2 -6343.696} C_VEL
LIN {X 0,Y 495.727,Z 359.736,A -85,B 0,C 180,E1 -6346.306,E2 -6346.306} C_VEL
LIN {X 0,Y 495.78,Z 359.728,A -85,B 0,C 180,E1 -6349.303,E2 -6349.303} C_VEL
LIN {X 0,Y 495.764,Z 359.731,A -85,B 0,C 180,E1 -6351.411,E2 -6351.411} C_VEL
LIN {X 0,Y 495.759,Z 359.729,A -85,B 0,C 180,E1 -6354.464,E2 -6354.464} C_VEL
LIN {X 0,Y 495.77,Z 359.731,A -85,B 0,C 180,E1 -6357.407,E2 -6357.407} C_VEL
LIN {X 0,Y 495.791,Z 359.727,A -85,B 0,C 180,E1 -6360.774,E2 -6360.774} C_VEL
LIN {X 0,Y 495.532,Z 360.389,A -85,B 0,C 180,E1 -6361.225,E2 -6361.225} C_VEL
LIN {X 0,Y 494.385,Z 362.959,A -85,B 0,C 180,E1 -6361.848,E2 -6361.848} C_VEL
LIN {X 0,Y 490.609,Z 370.011,A -85,B 0,C 180,E1 -6363.194,E2 -6363.194} C_VEL
LIN {X 0,Y 489.614,Z 372.898,A -85,B 0,C 180,E1 -6363.792,E2 -6363.792} C_VEL
LIN {X 0,Y 489.507,Z 373.846,A -85,B 0,C 180,E1 -6363.996,E2 -6363.996} C_VEL
LIN {X 0,Y 489.385,Z 377.516,A -85,B 0,C 180,E1 -6364.789,E2 -6364.789} C_VEL
LIN {X 0,Y 491.826,Z 389.48,A -85,B 0,C 180,E1 -6365.057,E2 -6365.057} C_VEL
LIN {X 0,Y 491.177,Z 484.278,A -85,B 0,C 180,E1 -6366.476,E2 -6366.476} C_VEL
LIN {X 0,Y 490.967,Z 497.514,A -85,B 0,C 180,E1 -6366.847,E2 -6366.847} C_VEL
LIN {X 0,Y 490.643,Z 509.91,A -85,B 0,C 180,E1 -6367.359,E2 -6367.359} C_VEL
LIN {X 0,Y 490.333,Z 521.475,A -85,B 0,C 180,E1 -6368.01,E2 -6368.01} C_VEL
LIN {X 0,Y 489.9,Z 533.153,A -85,B 0,C 180,E1 -6368.857,E2 -6368.857} C_VEL
LIN {X 0,Y 489.448,Z 543.945,A -85,B 0,C 180,E1 -6369.842,E2 -6369.842} C_VEL
LIN {X 0,Y 489.061,Z 553.366,A -85,B 0,C 180,E1 -6370.918,E2 -6370.918} C_VEL
LIN {X 0,Y 488.734,Z 561.184,A -85,B 0,C 180,E1 -6372.009,E2 -6372.009} C_VEL
LIN {X 0,Y 488.471,Z 568.575,A -85,B 0,C 180,E1 -6373.277,E2 -6373.277} C_VEL
LIN {X 0,Y 488.248,Z 574.994,A -85,B 0,C 180,E1 -6374.672,E2 -6374.672} C_VEL
LIN {X 0,Y 488.105,Z 579.171,A -85,B 0,C 180,E1 -6375.832,E2 -6375.832} C_VEL
LIN {X 0,Y 488.034,Z 581.596,A -85,B 0,C 180,E1 -6376.679,E2 -6376.679} C_VEL
LIN {X 0,Y 487.99,Z 583.57,A -85,B 0,C 180,E1 -6377.524,E2 -6377.524} C_VEL
LIN {X 0,Y 487.971,Z 585.116,A -85,B 0,C 180,E1 -6378.368,E2 -6378.368} C_VEL
LIN {X 0,Y 487.91,Z 586.196,A -85,B 0,C 180,E1 -6379.208,E2 -6379.208} C_VEL
LIN {X 0,Y 487.86,Z 587.155,A -85,B 0,C 180,E1 -6380.882,E2 -6380.882} C_VEL
LIN {X 0,Y 487.917,Z 587.044,A -85,B 0,C 180,E1 -6381.718,E2 -6381.718} C_VEL
LIN {X 0,Y 487.988,Z 585.563,A -85,B 0,C 180,E1 -6383.384,E2 -6383.384} C_VEL
LIN {X 0,Y 488.027,Z 584.239,A -85,B 0,C 180,E1 -6384.215,E2 -6384.215} C_VEL
LIN {X 0,Y 488.009,Z 581.452,A -85,B 0,C 180,E1 -6385.457,E2 -6385.457} C_VEL
LIN {X 0,Y 488.196,Z 577.643,A -85,B 0,C 180,E1 -6386.699,E2 -6386.699} C_VEL
LIN {X 0,Y 488.237,Z 572.751,A -85,B 0,C 180,E1 -6387.938,E2 -6387.938} C_VEL
LIN {X 0,Y 488.516,Z 566.592,A -85,B 0,C 180,E1 -6389.176,E2 -6389.176} C_VEL
LIN {X 0,Y 488.796,Z 558.927,A -85,B 0,C 180,E1 -6390.412,E2 -6390.412} C_VEL
LIN {X 0,Y 489.211,Z 549.357,A -85,B 0,C 180,E1 -6391.646,E2 -6391.646} C_VEL
LIN {X 0,Y 489.532,Z 539.509,A -85,B 0,C 180,E1 -6392.674,E2 -6392.674} C_VEL
LIN {X 0,Y 489.93,Z 528.368,A -85,B 0,C 180,E1 -6393.598,E2 -6393.598} C_VEL
LIN {X 0,Y 490.367,Z 517.453,A -85,B 0,C 180,E1 -6394.315,E2 -6394.315} C_VEL
LIN {X 0,Y 490.669,Z 505.405,A -85,B 0,C 180,E1 -6394.93,E2 -6394.93} C_VEL
LIN {X 0,Y 490.905,Z 492.755,A -85,B 0,C 180,E1 -6395.391,E2 -6395.391} C_VEL
LIN {X 0,Y 491.189,Z 479.302,A -85,B 0,C 180,E1 -6395.697,E2 -6395.697} C_VEL
LIN {X 0,Y 491.745,Z 388.453,A -85,B 0,C 180,E1 -6397.034,E2 -6397.034} C_VEL
LIN {X 0,Y 489.345,Z 377.343,A -85,B 0,C 180,E1 -6397.29,E2 -6397.29} C_VEL
LIN {X 0,Y 489.598,Z 367.088,A -85,B 0,C 180,E1 -6399.502,E2 -6399.502} C_VEL
LIN {X 0,Y 488.808,Z 360.6,A -85,B 0,C 180,E1 -6400.982,E2 -6400.982} C_VEL
LIN {X 0,Y 488.744,Z 360.607,A -85,B 0,C 180,E1 -6404.149,E2 -6404.149} C_VEL
LIN {X 0,Y 488.734,Z 360.606,A -85,B 0,C 180,E1 -6406.714,E2 -6406.714} C_VEL
LIN {X 0,Y 488.748,Z 360.6,A -85,B 0,C 180,E1 -6409.313,E2 -6409.313} C_VEL
LIN {X 0,Y 488.705,Z 360.609,A -85,B 0,C 180,E1 -6411.956,E2 -6411.956} C_VEL
LIN {X 0,Y 488.749,Z 360.601,A -85,B 0,C 180,E1 -6415.052,E2 -6415.052} C_VEL
LIN {X 0,Y 488.75,Z 360.601,A -85,B 0,C 180,E1 -6417.396,E2 -6417.396} C_VEL
LIN {X 0,Y 488.721,Z 360.609,A -85,B 0,C 180,E1 -6420.364,E2 -6420.364} C_VEL
LIN {X 0,Y 488.737,Z 360.604,A -85,B 0,C 180,E1 -6423.484,E2 -6423.484} C_VEL
LIN {X 0,Y 488.69,Z 360.612,A -85,B 0,C 180,E1 -6426.355,E2 -6426.355} C_VEL
LIN {X 0,Y 488.701,Z 360.608,A -85,B 0,C 180,E1 -6429.253,E2 -6429.253} C_VEL
LIN {X 0,Y 488.706,Z 360.609,A -85,B 0,C 180,E1 -6431.599,E2 -6431.599} C_VEL
LIN {X 0,Y 488.71,Z 360.607,A -85,B 0,C 180,E1 -6434.8,E2 -6434.8} C_VEL
LIN {X 0,Y 488.729,Z 360.607,A -85,B 0,C 180,E1 -6437.478,E2 -6437.478} C_VEL
LIN {X 0,Y 488.739,Z 360.603,A -85,B 0,C 180,E1 -6440.749,E2 -6440.749} C_VEL
LIN {X 0,Y 488.679,Z 360.616,A -85,B 0,C 180,E1 -6443.868,E2 -6443.868} C_VEL
LIN {X 0,Y 488.734,Z 360.604,A -85,B 0,C 180,E1 -6446.876,E2 -6446.876} C_VEL
LIN {X 0,Y 488.718,Z 360.611,A -85,B 0,C 180,E1 -6449.78,E2 -6449.78} C_VEL
LIN {X 0,Y 488.792,Z 360.599,A -85,B 0,C 180,E1 -6453.054,E2 -6453.054} C_VEL
LIN {X 0,Y 488.694,Z 360.609,A -85,B 0,C 180,E1 -6456.254,E2 -6456.254} C_VEL
LIN {X 0,Y 488.74,Z 360.606,A -85,B 0,C 180,E1 -6459.174,E2 -6459.174} C_VEL
LIN {X 0,Y 488.751,Z 360.606,A -85,B 0,C 180,E1 -6461.627,E2 -6461.627} C_VEL
LIN {X 0,Y 488.756,Z 360.605,A -85,B 0,C 180,E1 -6464.999,E2 -6464.999} C_VEL
LIN {X 0,Y 488.824,Z 360.593,A -85,B 0,C 180,E1 -6468.388,E2 -6468.388} C_VEL
LIN {X 0,Y 488.81,Z 360.596,A -85,B 0,C 180,E1 -6471.733,E2 -6471.733} C_VEL
LIN {X 0,Y 488.848,Z 360.59,A -85,B 0,C 180,E1 -6474.224,E2 -6474.224} C_VEL
LIN {X 0,Y 488.954,Z 360.579,A -85,B 0,C 180,E1 -6477.528,E2 -6477.528} C_VEL
LIN {X 0,Y 488.96,Z 360.576,A -85,B 0,C 180,E1 -6480,E2 -6480} C_VEL
LIN {X 0,Y 488.954,Z 360.579,A -85,B 0,C 180,E1 -6482.471,E2 -6482.471} C_VEL
LIN {X 0,Y 488.853,Z 360.589,A -85,B 0,C 180,E1 -6485.776,E2 -6485.776} C_VEL
LIN {X 0,Y 488.81,Z 360.596,A -85,B 0,C 180,E1 -6488.266,E2 -6488.266} C_VEL
LIN {X 0,Y 488.824,Z 360.593,A -85,B 0,C 180,E1 -6491.612,E2 -6491.612} C_VEL
LIN {X 0,Y 488.755,Z 360.604,A -85,B 0,C 180,E1 -6495,E2 -6495} C_VEL
LIN {X 0,Y 488.746,Z 360.608,A -85,B 0,C 180,E1 -6498.442,E2 -6498.442} C_VEL
LIN {X 0,Y 488.732,Z 360.607,A -85,B 0,C 180,E1 -6501.07,E2 -6501.07} C_VEL
LIN {X 0,Y 488.693,Z 360.609,A -85,B 0,C 180,E1 -6503.745,E2 -6503.745} C_VEL
LIN {X 0,Y 488.791,Z 360.599,A -85,B 0,C 180,E1 -6506.946,E2 -6506.946} C_VEL
LIN {X 0,Y 488.703,Z 360.613,A -85,B 0,C 180,E1 -6510.364,E2 -6510.364} C_VEL
LIN {X 0,Y 488.729,Z 360.604,A -85,B 0,C 180,E1 -6513.485,E2 -6513.485} C_VEL
LIN {X 0,Y 488.684,Z 360.614,A -85,B 0,C 180,E1 -6516.356,E2 -6516.356} C_VEL
LIN {X 0,Y 488.737,Z 360.603,A -85,B 0,C 180,E1 -6519.251,E2 -6519.251} C_VEL
LIN {X 0,Y 488.726,Z 360.607,A -85,B 0,C 180,E1 -6522.522,E2 -6522.522} C_VEL
LIN {X 0,Y 488.707,Z 360.606,A -85,B 0,C 180,E1 -6525.199,E2 -6525.199} C_VEL
LIN {X 0,Y 488.705,Z 360.609,A -85,B 0,C 180,E1 -6528.401,E2 -6528.401} C_VEL
LIN {X 0,Y 488.702,Z 360.607,A -85,B 0,C 180,E1 -6530.948,E2 -6530.948} C_VEL
LIN {X 0,Y 488.684,Z 360.615,A -85,B 0,C 180,E1 -6533.869,E2 -6533.869} C_VEL
LIN {X 0,Y 488.738,Z 360.602,A -85,B 0,C 180,E1 -6536.878,E2 -6536.878} C_VEL
LIN {X 0,Y 488.734,Z 360.609,A -85,B 0,C 180,E1 -6539.782,E2 -6539.782} C_VEL
LIN {X 0,Y 488.792,Z 360.598,A -85,B 0,C 180,E1 -6543.057,E2 -6543.057} C_VEL
LIN {X 0,Y 488.796,Z 360.772,A -85,B 0,C 180,E1 -6544.047,E2 -6544.047} C_VEL
LIN {X 0,Y 490.813,Z 371.4,A -85,B 0,C 180,E1 -6545.915,E2 -6545.915} C_VEL
LIN {X 0,Y 490.381,Z 387.292,A -85,B 0,C 180,E1 -6548.511,E2 -6548.511} C_VEL
LIN {X 0,Y 489.608,Z 409.142,A -85,B 0,C 180,E1 -6552.024,E2 -6552.024} C_VEL
LIN {X 0,Y 489.271,Z 419.963,A -85,B 0,C 180,E1 -6553.734,E2 -6553.734} C_VEL
LIN {X 0,Y 491.677,Z 437.064,A -85,B 0,C 180,E1 -6554.066,E2 -6554.066} C_VEL
LIN {X 0,Y 491.102,Z 528.206,A -85,B 0,C 180,E1 -6555.418,E2 -6555.418} C_VEL
LIN {X 0,Y 490.784,Z 541.574,A -85,B 0,C 180,E1 -6555.779,E2 -6555.779} C_VEL
LIN {X 0,Y 490.385,Z 553.795,A -85,B 0,C 180,E1 -6556.269,E2 -6556.269} C_VEL
LIN {X 0,Y 489.995,Z 566.133,A -85,B 0,C 180,E1 -6556.945,E2 -6556.945} C_VEL
LIN {X 0,Y 489.539,Z 577.769,A -85,B 0,C 180,E1 -6557.775,E2 -6557.775} C_VEL
LIN {X 0,Y 489.162,Z 588.25,A -85,B 0,C 180,E1 -6558.711,E2 -6558.711} C_VEL
LIN {X 0,Y 488.845,Z 596.822,A -85,B 0,C 180,E1 -6559.647,E2 -6559.647} C_VEL
LIN {X 0,Y 488.498,Z 604.73,A -85,B 0,C 180,E1 -6560.686,E2 -6560.686} C_VEL
LIN {X 0,Y 488.277,Z 612.461,A -85,B 0,C 180,E1 -6561.933,E2 -6561.933} C_VEL
LIN {X 0,Y 488.1,Z 619.587,A -85,B 0,C 180,E1 -6563.386,E2 -6563.386} C_VEL
LIN {X 0,Y 488.019,Z 624.329,A -85,B 0,C 180,E1 -6564.629,E2 -6564.629} C_VEL
LIN {X 0,Y 487.948,Z 627.952,A -85,B 0,C 180,E1 -6565.87,E2 -6565.87} C_VEL
LIN {X 0,Y 487.969,Z 629.823,A -85,B 0,C 180,E1 -6566.697,E2 -6566.697} C_VEL
LIN {X 0,Y 487.932,Z 631.223,A -85,B 0,C 180,E1 -6567.523,E2 -6567.523} C_VEL
LIN {X 0,Y 487.892,Z 632.221,A -85,B 0,C 180,E1 -6568.349,E2 -6568.349} C_VEL
LIN {X 0,Y 487.822,Z 633.042,A -85,B 0,C 180,E1 -6570,E2 -6570} C_VEL
LIN {X 0,Y 487.892,Z 632.213,A -85,B 0,C 180,E1 -6571.651,E2 -6571.651} C_VEL
LIN {X 0,Y 487.932,Z 631.212,A -85,B 0,C 180,E1 -6572.477,E2 -6572.477} C_VEL
LIN {X 0,Y 487.969,Z 629.808,A -85,B 0,C 180,E1 -6573.303,E2 -6573.303} C_VEL
LIN {X 0,Y 487.921,Z 626.852,A -85,B 0,C 180,E1 -6574.544,E2 -6574.544} C_VEL
LIN {X 0,Y 488.024,Z 622.858,A -85,B 0,C 180,E1 -6575.785,E2 -6575.785} C_VEL
LIN {X 0,Y 488.181,Z 616.716,A -85,B 0,C 180,E1 -6577.236,E2 -6577.236} C_VEL
LIN {X 0,Y 488.357,Z 610.006,A -85,B 0,C 180,E1 -6578.482,E2 -6578.482} C_VEL
LIN {X 0,Y 488.618,Z 601.685,A -85,B 0,C 180,E1 -6579.73,E2 -6579.73} C_VEL
LIN {X 0,Y 488.987,Z 593.162,A -85,B 0,C 180,E1 -6580.768,E2 -6580.768} C_VEL
LIN {X 0,Y 489.44,Z 582.64,A -85,B 0,C 180,E1 -6581.807,E2 -6581.807} C_VEL
LIN {X 0,Y 489.769,Z 571.091,A -85,B 0,C 180,E1 -6582.724,E2 -6582.724} C_VEL
LIN {X 0,Y 490.227,Z 558.902,A -85,B 0,C 180,E1 -6583.471,E2 -6583.471} C_VEL
LIN {X 0,Y 490.613,Z 546.532,A -85,B 0,C 180,E1 -6584.041,E2 -6584.041} C_VEL
LIN {X 0,Y 490.988,Z 533.846,A -85,B 0,C 180,E1 -6584.454,E2 -6584.454} C_VEL
LIN {X 0,Y 491.177,Z 518.826,A -85,B 0,C 180,E1 -6584.739,E2 -6584.739} C_VEL
LIN {X 0,Y 491.61,Z 435.142,A -85,B 0,C 180,E1 -6585.971,E2 -6585.971} C_VEL
LIN {X 0,Y 489.265,Z 419.593,A -85,B 0,C 180,E1 -6586.309,E2 -6586.309} C_VEL
LIN {X 0,Y 489.857,Z 401.178,A -85,B 0,C 180,E1 -6589.267,E2 -6589.267} C_VEL
LIN {X 0,Y 490.526,Z 383.857,A -85,B 0,C 180,E1 -6592.092,E2 -6592.092} C_VEL
LIN {X 0,Y 490.962,Z 371.883,A -85,B 0,C 180,E1 -6594.077,E2 -6594.077} C_VEL
LIN {X 0,Y 488.784,Z 360.604,A -85,B 0,C 180,E1 -6596.125,E2 -6596.125} C_VEL
LIN {X 0,Y 488.734,Z 360.604,A -85,B 0,C 180,E1 -6599.269,E2 -6599.269} C_VEL
LIN {X 0,Y 488.705,Z 360.612,A -85,B 0,C 180,E1 -6602.146,E2 -6602.146} C_VEL
LIN {X 0,Y 488.721,Z 360.605,A -85,B 0,C 180,E1 -6605.114,E2 -6605.114} C_VEL
LIN {X 0,Y 488.678,Z 360.613,A -85,B 0,C 180,E1 -6608.199,E2 -6608.199} C_VEL
LIN {X 0,Y 488.714,Z 360.606,A -85,B 0,C 180,E1 -6610.344,E2 -6610.344} C_VEL
LIN {X 0,Y 488.682,Z 360.613,A -85,B 0,C 180,E1 -6613.654,E2 -6613.654} C_VEL
LIN {X 0,Y 488.712,Z 360.604,A -85,B 0,C 180,E1 -6616.348,E2 -6616.348} C_VEL
LIN {X 0,Y 488.728,Z 360.608,A -85,B 0,C 180,E1 -6619.676,E2 -6619.676} C_VEL
LIN {X 0,Y 488.674,Z 360.609,A -85,B 0,C 180,E1 -6622.277,E2 -6622.277} C_VEL
LIN {X 0,Y 488.722,Z 360.605,A -85,B 0,C 180,E1 -6625.051,E2 -6625.051} C_VEL
LIN {X 0,Y 488.699,Z 360.608,A -85,B 0,C 180,E1 -6628.045,E2 -6628.045} C_VEL
LIN {X 0,Y 488.726,Z 360.603,A -85,B 0,C 180,E1 -6630.73,E2 -6630.73} C_VEL
LIN {X 0,Y 488.758,Z 360.598,A -85,B 0,C 180,E1 -6633.528,E2 -6633.528} C_VEL
LIN {X 0,Y 488.693,Z 360.602,A -85,B 0,C 180,E1 -6636.255,E2 -6636.255} C_VEL
LIN {X 0,Y 488.739,Z 360.608,A -85,B 0,C 180,E1 -6639.175,E2 -6639.175} C_VEL
LIN {X 0,Y 488.75,Z 360.603,A -85,B 0,C 180,E1 -6641.627,E2 -6641.627} C_VEL
LIN {X 0,Y 488.752,Z 360.604,A -85,B 0,C 180,E1 -6644.999,E2 -6644.999} C_VEL
LIN {X 0,Y 488.825,Z 360.591,A -85,B 0,C 180,E1 -6648.388,E2 -6648.388} C_VEL
LIN {X 0,Y 488.81,Z 360.593,A -85,B 0,C 180,E1 -6651.734,E2 -6651.734} C_VEL
LIN {X 0,Y 488.847,Z 360.585,A -85,B 0,C 180,E1 -6654.224,E2 -6654.224} C_VEL
LIN {X 0,Y 488.954,Z 360.574,A -85,B 0,C 180,E1 -6657.529,E2 -6657.529} C_VEL
LIN {X 0,Y 488.96,Z 360.573,A -85,B 0,C 180,E1 -6660,E2 -6660} C_VEL
LIN {X 0,Y 488.954,Z 360.578,A -85,B 0,C 180,E1 -6662.472,E2 -6662.472} C_VEL
LIN {X 0,Y 488.848,Z 360.588,A -85,B 0,C 180,E1 -6665.776,E2 -6665.776} C_VEL
LIN {X 0,Y 488.81,Z 360.593,A -85,B 0,C 180,E1 -6668.267,E2 -6668.267} C_VEL
LIN {X 0,Y 488.799,Z 360.593,A -85,B 0,C 180,E1 -6671.613,E2 -6671.613} C_VEL
LIN {X 0,Y 488.756,Z 360.602,A -85,B 0,C 180,E1 -6675.001,E2 -6675.001} C_VEL
LIN {X 0,Y 488.747,Z 360.607,A -85,B 0,C 180,E1 -6678.443,E2 -6678.443} C_VEL
LIN {X 0,Y 488.7,Z 360.606,A -85,B 0,C 180,E1 -6681.071,E2 -6681.071} C_VEL
LIN {X 0,Y 488.687,Z 360.609,A -85,B 0,C 180,E1 -6683.746,E2 -6683.746} C_VEL
LIN {X 0,Y 488.792,Z 360.59,A -85,B 0,C 180,E1 -6686.946,E2 -6686.946} C_VEL
LIN {X 0,Y 488.704,Z 360.611,A -85,B 0,C 180,E1 -6690.364,E2 -6690.364} C_VEL
LIN {X 0,Y 488.731,Z 360.603,A -85,B 0,C 180,E1 -6693.485,E2 -6693.485} C_VEL
LIN {X 0,Y 488.685,Z 360.613,A -85,B 0,C 180,E1 -6696.357,E2 -6696.357} C_VEL
LIN {X 0,Y 488.739,Z 360.602,A -85,B 0,C 180,E1 -6699.251,E2 -6699.251} C_VEL
LIN {X 0,Y 488.729,Z 360.605,A -85,B 0,C 180,E1 -6702.522,E2 -6702.522} C_VEL
LIN {X 0,Y 488.71,Z 360.609,A -85,B 0,C 180,E1 -6705.2,E2 -6705.2} C_VEL
LIN {X 0,Y 488.711,Z 360.61,A -85,B 0,C 180,E1 -6708.4,E2 -6708.4} C_VEL
LIN {X 0,Y 488.747,Z 360.602,A -85,B 0,C 180,E1 -6710.942,E2 -6710.942} C_VEL
LIN {X 0,Y 488.687,Z 360.614,A -85,B 0,C 180,E1 -6713.87,E2 -6713.87} C_VEL
LIN {X 0,Y 488.74,Z 360.603,A -85,B 0,C 180,E1 -6716.878,E2 -6716.878} C_VEL
LIN {X 0,Y 488.736,Z 360.609,A -85,B 0,C 180,E1 -6719.782,E2 -6719.782} C_VEL
LIN {X 0,Y 488.781,Z 360.682,A -85,B 0,C 180,E1 -6721.046,E2 -6721.046} C_VEL
LIN {X 0,Y 489.72,Z 366.683,A -85,B 0,C 180,E1 -6722.431,E2 -6722.431} C_VEL
LIN {X 0,Y 489.507,Z 373.846,A -85,B 0,C 180,E1 -6723.996,E2 -6723.996} C_VEL
LIN {X 0,Y 489.181,Z 376.245,A -85,B 0,C 180,E1 -6724.335,E2 -6724.335} C_VEL
LIN {X 0,Y 488.512,Z 379.403,A -85,B 0,C 180,E1 -6724.577,E2 -6724.577} C_VEL
LIN {X 0,Y 487.259,Z 384.906,A -85,B 0,C 180,E1 -6724.795,E2 -6724.795} C_VEL
LIN {X 0,Y 485.15,Z 397.446,A -85,B 0,C 180,E1 -6724.932,E2 -6724.932} C_VEL
LIN {X 0,Y 485.019,Z 403.879,A -85,B 0,C 180,E1 -6725.029,E2 -6725.029} C_VEL
LIN {X 0,Y 484.341,Z 484.893,A -85,B 0,C 180,E1 -6726.262,E2 -6726.262} C_VEL
LIN {X 0,Y 484.123,Z 497.676,A -85,B 0,C 180,E1 -6726.626,E2 -6726.626} C_VEL
LIN {X 0,Y 483.791,Z 509.848,A -85,B 0,C 180,E1 -6727.133,E2 -6727.133} C_VEL
LIN {X 0,Y 483.459,Z 521.525,A -85,B 0,C 180,E1 -6727.793,E2 -6727.793} C_VEL
LIN {X 0,Y 482.995,Z 533.442,A -85,B 0,C 180,E1 -6728.668,E2 -6728.668} C_VEL
LIN {X 0,Y 482.528,Z 544.082,A -85,B 0,C 180,E1 -6729.651,E2 -6729.651} C_VEL
LIN {X 0,Y 482.13,Z 552.695,A -85,B 0,C 180,E1 -6730.633,E2 -6730.633} C_VEL
LIN {X 0,Y 481.744,Z 561.102,A -85,B 0,C 180,E1 -6731.806,E2 -6731.806} C_VEL
LIN {X 0,Y 481.466,Z 568.216,A -85,B 0,C 180,E1 -6733.026,E2 -6733.026} C_VEL
LIN {X 0,Y 481.214,Z 574.181,A -85,B 0,C 180,E1 -6734.296,E2 -6734.296} C_VEL
LIN {X 0,Y 481.05,Z 579.07,A -85,B 0,C 180,E1 -6735.62,E2 -6735.62} C_VEL
LIN {X 0,Y 480.93,Z 582.674,A -85,B 0,C 180,E1 -6736.909,E2 -6736.909} C_VEL
LIN {X 0,Y 480.889,Z 585.39,A -85,B 0,C 180,E1 -6738.29,E2 -6738.29} C_VEL
LIN {X 0,Y 480.788,Z 587.129,A -85,B 0,C 180,E1 -6739.898,E2 -6739.898} C_VEL
LIN {X 0,Y 480.815,Z 587.41,A -85,B 0,C 180,E1 -6741.595,E2 -6741.595} C_VEL
LIN {X 0,Y 480.843,Z 586.956,A -85,B 0,C 180,E1 -6742.441,E2 -6742.441} C_VEL
LIN {X 0,Y 480.942,Z 584.794,A -85,B 0,C 180,E1 -6744.129,E2 -6744.129} C_VEL
LIN {X 0,Y 480.911,Z 582.111,A -85,B 0,C 180,E1 -6745.39,E2 -6745.39} C_VEL
LIN {X 0,Y 481.119,Z 578.41,A -85,B 0,C 180,E1 -6746.65,E2 -6746.65} C_VEL
LIN {X 0,Y 481.178,Z 573.629,A -85,B 0,C 180,E1 -6747.907,E2 -6747.907} C_VEL
LIN {X 0,Y 481.436,Z 567.597,A -85,B 0,C 180,E1 -6749.164,E2 -6749.164} C_VEL
LIN {X 0,Y 481.757,Z 560.12,A -85,B 0,C 180,E1 -6750.418,E2 -6750.418} C_VEL
LIN {X 0,Y 482.094,Z 552.488,A -85,B 0,C 180,E1 -6751.462,E2 -6751.462} C_VEL
LIN {X 0,Y 482.471,Z 542.159,A -85,B 0,C 180,E1 -6752.609,E2 -6752.609} C_VEL
LIN {X 0,Y 482.879,Z 531.658,A -85,B 0,C 180,E1 -6753.546,E2 -6753.546} C_VEL
LIN {X 0,Y 483.278,Z 521.509,A -85,B 0,C 180,E1 -6754.274,E2 -6754.274} C_VEL
LIN {X 0,Y 483.641,Z 510.553,A -85,B 0,C 180,E1 -6754.897,E2 -6754.897} C_VEL
LIN {X 0,Y 483.932,Z 497.588,A -85,B 0,C 180,E1 -6755.443,E2 -6755.443} C_VEL
LIN {X 0,Y 484.185,Z 484.736,A -85,B 0,C 180,E1 -6755.805,E2 -6755.805} C_VEL
LIN {X 0,Y 484.798,Z 414.828,A -85,B 0,C 180,E1 -6756.865,E2 -6756.865} C_VEL
LIN {X 0,Y 484.877,Z 389.171,A -85,B 0,C 180,E1 -6757.25,E2 -6757.25} C_VEL
LIN {X 0,Y 482.379,Z 377.582,A -85,B 0,C 180,E1 -6757.534,E2 -6757.534} C_VEL
LIN {X 0,Y 482.615,Z 367.914,A -85,B 0,C 180,E1 -6759.64,E2 -6759.64} C_VEL
LIN {X 0,Y 481.794,Z 361.473,A -85,B 0,C 180,E1 -6761.144,E2 -6761.144} C_VEL
LIN {X 0,Y 481.696,Z 361.487,A -85,B 0,C 180,E1 -6764.361,E2 -6764.361} C_VEL
LIN {X 0,Y 481.694,Z 361.48,A -85,B 0,C 180,E1 -6766.966,E2 -6766.966} C_VEL
LIN {X 0,Y 481.71,Z 361.478,A -85,B 0,C 180,E1 -6769.606,E2 -6769.606} C_VEL
LIN {X 0,Y 481.658,Z 361.491,A -85,B 0,C 180,E1 -6772.294,E2 -6772.294} C_VEL
LIN {X 0,Y 481.715,Z 361.477,A -85,B 0,C 180,E1 -6775.236,E2 -6775.236} C_VEL
LIN {X 0,Y 481.704,Z 361.481,A -85,B 0,C 180,E1 -6777.831,E2 -6777.831} C_VEL
LIN {X 0,Y 481.654,Z 361.486,A -85,B 0,C 180,E1 -6780.71,E2 -6780.71} C_VEL
LIN {X 0,Y 481.698,Z 361.482,A -85,B 0,C 180,E1 -6783.732,E2 -6783.732} C_VEL
LIN {X 0,Y 481.63,Z 361.489,A -85,B 0,C 180,E1 -6786.746,E2 -6786.746} C_VEL
LIN {X 0,Y 481.676,Z 361.487,A -85,B 0,C 180,E1 -6789.939,E2 -6789.939} C_VEL
LIN {X 0,Y 481.637,Z 361.489,A -85,B 0,C 180,E1 -6793.299,E2 -6793.299} C_VEL
LIN {X 0,Y 481.681,Z 361.482,A -85,B 0,C 180,E1 -6796.704,E2 -6796.704} C_VEL
LIN {X 0,Y 481.685,Z 361.486,A -85,B 0,C 180,E1 -6800.06,E2 -6800.06} C_VEL
LIN {X 0,Y 481.624,Z 361.492,A -85,B 0,C 180,E1 -6803.252,E2 -6803.252} C_VEL
LIN {X 0,Y 481.705,Z 361.481,A -85,B 0,C 180,E1 -6806.329,E2 -6806.329} C_VEL
LIN {X 0,Y 481.645,Z 361.489,A -85,B 0,C 180,E1 -6809.416,E2 -6809.416} C_VEL
LIN {X 0,Y 481.696,Z 361.482,A -85,B 0,C 180,E1 -6812.167,E2 -6812.167} C_VEL
LIN {X 0,Y 481.713,Z 361.481,A -85,B 0,C 180,E1 -6814.969,E2 -6814.969} C_VEL
LIN {X 0,Y 481.653,Z 361.491,A -85,B 0,C 180,E1 -6817.705,E2 -6817.705} C_VEL
LIN {X 0,Y 481.701,Z 361.481,A -85,B 0,C 180,E1 -6820.392,E2 -6820.392} C_VEL
LIN {X 0,Y 481.684,Z 361.485,A -85,B 0,C 180,E1 -6823.033,E2 -6823.033} C_VEL
LIN {X 0,Y 481.688,Z 361.486,A -85,B 0,C 180,E1 -6825.638,E2 -6825.638} C_VEL
LIN {X 0,Y 481.787,Z 361.47,A -85,B 0,C 180,E1 -6828.216,E2 -6828.216} C_VEL
LIN {X 0,Y 481.755,Z 361.477,A -85,B 0,C 180,E1 -6831.611,E2 -6831.611} C_VEL
LIN {X 0,Y 481.808,Z 361.467,A -85,B 0,C 180,E1 -6834.139,E2 -6834.139} C_VEL
LIN {X 0,Y 481.921,Z 361.456,A -85,B 0,C 180,E1 -6837.492,E2 -6837.492} C_VEL
LIN {X 0,Y 481.931,Z 361.452,A -85,B 0,C 180,E1 -6840,E2 -6840} C_VEL
LIN {X 0,Y 481.921,Z 361.456,A -85,B 0,C 180,E1 -6842.507,E2 -6842.507} C_VEL
LIN {X 0,Y 481.813,Z 361.467,A -85,B 0,C 180,E1 -6845.86,E2 -6845.86} C_VEL
LIN {X 0,Y 481.755,Z 361.476,A -85,B 0,C 180,E1 -6848.388,E2 -6848.388} C_VEL
LIN {X 0,Y 481.787,Z 361.47,A -85,B 0,C 180,E1 -6851.784,E2 -6851.784} C_VEL
LIN {X 0,Y 481.735,Z 361.478,A -85,B 0,C 180,E1 -6855.224,E2 -6855.224} C_VEL
LIN {X 0,Y 481.703,Z 361.483,A -85,B 0,C 180,E1 -6858.722,E2 -6858.722} C_VEL
LIN {X 0,Y 481.663,Z 361.485,A -85,B 0,C 180,E1 -6861.394,E2 -6861.394} C_VEL
LIN {X 0,Y 481.674,Z 361.486,A -85,B 0,C 180,E1 -6864.113,E2 -6864.113} C_VEL
LIN {X 0,Y 481.744,Z 361.476,A -85,B 0,C 180,E1 -6867.141,E2 -6867.141} C_VEL
LIN {X 0,Y 481.671,Z 361.484,A -85,B 0,C 180,E1 -6869.742,E2 -6869.742} C_VEL
LIN {X 0,Y 481.666,Z 361.486,A -85,B 0,C 180,E1 -6872.675,E2 -6872.675} C_VEL
LIN {X 0,Y 481.637,Z 361.489,A -85,B 0,C 180,E1 -6875.71,E2 -6875.71} C_VEL
LIN {X 0,Y 481.709,Z 361.478,A -85,B 0,C 180,E1 -6879.354,E2 -6879.354} C_VEL
LIN {X 0,Y 481.668,Z 361.489,A -85,B 0,C 180,E1 -6882.159,E2 -6882.159} C_VEL
LIN {X 0,Y 481.655,Z 361.488,A -85,B 0,C 180,E1 -6884.458,E2 -6884.458} C_VEL
LIN {X 0,Y 481.644,Z 361.49,A -85,B 0,C 180,E1 -6887.84,E2 -6887.84} C_VEL
LIN {X 0,Y 481.678,Z 361.483,A -85,B 0,C 180,E1 -6890.652,E2 -6890.652} C_VEL
LIN {X 0,Y 481.63,Z 361.488,A -85,B 0,C 180,E1 -6893.376,E2 -6893.376} C_VEL
LIN {X 0,Y 481.708,Z 361.48,A -85,B 0,C 180,E1 -6896.331,E2 -6896.331} C_VEL
LIN {X 0,Y 481.658,Z 361.486,A -85,B 0,C 180,E1 -6899.416,E2 -6899.416} C_VEL
LIN {X 0,Y 481.701,Z 361.485,A -85,B 0,C 180,E1 -6902.169,E2 -6902.169} C_VEL
LIN {X 0,Y 481.75,Z 361.68,A -85,B 0,C 180,E1 -6903.872,E2 -6903.872} C_VEL
LIN {X 0,Y 483.825,Z 372.339,A -85,B 0,C 180,E1 -6905.773,E2 -6905.773} C_VEL
LIN {X 0,Y 483.626,Z 381.812,A -85,B 0,C 180,E1 -6907.351,E2 -6907.351} C_VEL
LIN {X 0,Y 482.891,Z 400.69,A -85,B 0,C 180,E1 -6910.444,E2 -6910.444} C_VEL
LIN {X 0,Y 482.318,Z 418.008,A -85,B 0,C 180,E1 -6913.253,E2 -6913.253} C_VEL
LIN {X 0,Y 482.28,Z 419.514,A -85,B 0,C 180,E1 -6913.497,E2 -6913.497} C_VEL
LIN {X 0,Y 484.83,Z 437.171,A -85,B 0,C 180,E1 -6913.85,E2 -6913.85} C_VEL
LIN {X 0,Y 484.21,Z 528.758,A -85,B 0,C 180,E1 -6915.232,E2 -6915.232} C_VEL
LIN {X 0,Y 483.872,Z 541.838,A -85,B 0,C 180,E1 -6915.598,E2 -6915.598} C_VEL
LIN {X 0,Y 483.43,Z 554.479,A -85,B 0,C 180,E1 -6916.121,E2 -6916.121} C_VEL
LIN {X 0,Y 483.053,Z 565.729,A -85,B 0,C 180,E1 -6916.754,E2 -6916.754} C_VEL
LIN {X 0,Y 482.56,Z 577.485,A -85,B 0,C 180,E1 -6917.603,E2 -6917.603} C_VEL
LIN {X 0,Y 482.184,Z 587.89,A -85,B 0,C 180,E1 -6918.546,E2 -6918.546} C_VEL
LIN {X 0,Y 481.821,Z 596.471,A -85,B 0,C 180,E1 -6919.495,E2 -6919.495} C_VEL
LIN {X 0,Y 481.463,Z 604.386,A -85,B 0,C 180,E1 -6920.548,E2 -6920.548} C_VEL
LIN {X 0,Y 481.203,Z 612.121,A -85,B 0,C 180,E1 -6921.813,E2 -6921.813} C_VEL
LIN {X 0,Y 481.019,Z 619.251,A -85,B 0,C 180,E1 -6923.288,E2 -6923.288} C_VEL
LIN {X 0,Y 480.932,Z 623.996,A -85,B 0,C 180,E1 -6924.55,E2 -6924.55} C_VEL
LIN {X 0,Y 480.844,Z 627.618,A -85,B 0,C 180,E1 -6925.809,E2 -6925.809} C_VEL
LIN {X 0,Y 480.893,Z 629.491,A -85,B 0,C 180,E1 -6926.649,E2 -6926.649} C_VEL
LIN {X 0,Y 480.845,Z 630.891,A -85,B 0,C 180,E1 -6927.487,E2 -6927.487} C_VEL
LIN {X 0,Y 480.823,Z 631.889,A -85,B 0,C 180,E1 -6928.325,E2 -6928.325} C_VEL
LIN {X 0,Y 480.745,Z 632.709,A -85,B 0,C 180,E1 -6930,E2 -6930} C_VEL
LIN {X 0,Y 480.823,Z 631.88,A -85,B 0,C 180,E1 -6931.675,E2 -6931.675} C_VEL
LIN {X 0,Y 480.845,Z 630.877,A -85,B 0,C 180,E1 -6932.513,E2 -6932.513} C_VEL
LIN {X 0,Y 480.893,Z 629.473,A -85,B 0,C 180,E1 -6933.351,E2 -6933.351} C_VEL
LIN {X 0,Y 480.84,Z 626.515,A -85,B 0,C 180,E1 -6934.611,E2 -6934.611} C_VEL
LIN {X 0,Y 480.928,Z 622.52,A -85,B 0,C 180,E1 -6935.871,E2 -6935.871} C_VEL
LIN {X 0,Y 481.106,Z 616.38,A -85,B 0,C 180,E1 -6937.343,E2 -6937.343} C_VEL
LIN {X 0,Y 481.3,Z 609.672,A -85,B 0,C 180,E1 -6938.608,E2 -6938.608} C_VEL
LIN {X 0,Y 481.573,Z 601.354,A -85,B 0,C 180,E1 -6939.874,E2 -6939.874} C_VEL
LIN {X 0,Y 481.991,Z 592.847,A -85,B 0,C 180,E1 -6940.927,E2 -6940.927} C_VEL
LIN {X 0,Y 482.45,Z 582.406,A -85,B 0,C 180,E1 -6941.975,E2 -6941.975} C_VEL
LIN {X 0,Y 482.827,Z 570.67,A -85,B 0,C 180,E1 -6942.921,E2 -6942.921} C_VEL
LIN {X 0,Y 483.31,Z 558.665,A -85,B 0,C 180,E1 -6943.668,E2 -6943.668} C_VEL
LIN {X 0,Y 483.714,Z 546.355,A -85,B 0,C 180,E1 -6944.246,E2 -6944.246} C_VEL
LIN {X 0,Y 484.125,Z 533.764,A -85,B 0,C 180,E1 -6944.663,E2 -6944.663} C_VEL
LIN {X 0,Y 484.337,Z 520.793,A -85,B 0,C 180,E1 -6944.925,E2 -6944.925} C_VEL
LIN {X 0,Y 484.724,Z 435.6,A -85,B 0,C 180,E1 -6946.202,E2 -6946.202} C_VEL
LIN {X 0,Y 482.263,Z 419.249,A -85,B 0,C 180,E1 -6946.564,E2 -6946.564} C_VEL
LIN {X 0,Y 482.943,Z 400.959,A -85,B 0,C 180,E1 -6949.554,E2 -6949.554} C_VEL
LIN {X 0,Y 483.696,Z 382.352,A -85,B 0,C 180,E1 -6952.646,E2 -6952.646} C_VEL
LIN {X 0,Y 484.01,Z 373.061,A -85,B 0,C 180,E1 -6954.217,E2 -6954.217} C_VEL
LIN {X 0,Y 481.75,Z 361.48,A -85,B 0,C 180,E1 -6956.361,E2 -6956.361} C_VEL
LIN {X 0,Y 481.688,Z 361.483,A -85,B 0,C 180,E1 -6959.74,E2 -6959.74} C_VEL
LIN {X 0,Y 481.672,Z 361.484,A -85,B 0,C 180,E1 -6962.673,E2 -6962.673} C_VEL
LIN {X 0,Y 481.641,Z 361.492,A -85,B 0,C 180,E1 -6965.708,E2 -6965.708} C_VEL
LIN {X 0,Y 481.668,Z 361.482,A -85,B 0,C 180,E1 -6968.858,E2 -6968.858} C_VEL
LIN {X 0,Y 481.649,Z 361.49,A -85,B 0,C 180,E1 -6971.912,E2 -6971.912} C_VEL
LIN {X 0,Y 481.655,Z 361.483,A -85,B 0,C 180,E1 -6974.457,E2 -6974.457} C_VEL
LIN {X 0,Y 481.683,Z 361.478,A -85,B 0,C 180,E1 -6976.845,E2 -6976.845} C_VEL
LIN {X 0,Y 481.684,Z 361.482,A -85,B 0,C 180,E1 -6980.06,E2 -6980.06} C_VEL
LIN {X 0,Y 481.624,Z 361.49,A -85,B 0,C 180,E1 -6983.253,E2 -6983.253} C_VEL
LIN {X 0,Y 481.703,Z 361.478,A -85,B 0,C 180,E1 -6986.329,E2 -6986.329} C_VEL
LIN {X 0,Y 481.652,Z 361.49,A -85,B 0,C 180,E1 -6989.415,E2 -6989.415} C_VEL
LIN {X 0,Y 481.695,Z 361.479,A -85,B 0,C 180,E1 -6992.168,E2 -6992.168} C_VEL
LIN {X 0,Y 481.711,Z 361.471,A -85,B 0,C 180,E1 -6994.97,E2 -6994.97} C_VEL
LIN {X 0,Y 481.652,Z 361.487,A -85,B 0,C 180,E1 -6997.705,E2 -6997.705} C_VEL
LIN {X 0,Y 481.699,Z 361.477,A -85,B 0,C 180,E1 -7000.393,E2 -7000.393} C_VEL
LIN {X 0,Y 481.683,Z 361.486,A -85,B 0,C 180,E1 -7003.034,E2 -7003.034} C_VEL
LIN {X 0,Y 481.682,Z 361.482,A -85,B 0,C 180,E1 -7005.639,E2 -7005.639} C_VEL
LIN {X 0,Y 481.787,Z 361.467,A -85,B 0,C 180,E1 -7008.216,E2 -7008.216} C_VEL
LIN {X 0,Y 481.755,Z 361.473,A -85,B 0,C 180,E1 -7011.612,E2 -7011.612} C_VEL
LIN {X 0,Y 481.808,Z 361.461,A -85,B 0,C 180,E1 -7014.14,E2 -7014.14} C_VEL
LIN {X 0,Y 481.921,Z 361.451,A -85,B 0,C 180,E1 -7017.493,E2 -7017.493} C_VEL
LIN {X 0,Y 481.931,Z 361.448,A -85,B 0,C 180,E1 -7020,E2 -7020} C_VEL
LIN {X 0,Y 481.921,Z 361.455,A -85,B 0,C 180,E1 -7022.508,E2 -7022.508} C_VEL
LIN {X 0,Y 481.809,Z 361.465,A -85,B 0,C 180,E1 -7025.861,E2 -7025.861} C_VEL
LIN {X 0,Y 481.755,Z 361.473,A -85,B 0,C 180,E1 -7028.389,E2 -7028.389} C_VEL
LIN {X 0,Y 481.744,Z 361.472,A -85,B 0,C 180,E1 -7031.785,E2 -7031.785} C_VEL
LIN {X 0,Y 481.736,Z 361.475,A -85,B 0,C 180,E1 -7035.225,E2 -7035.225} C_VEL
LIN {X 0,Y 481.705,Z 361.483,A -85,B 0,C 180,E1 -7038.722,E2 -7038.722} C_VEL
LIN {X 0,Y 481.64,Z 361.484,A -85,B 0,C 180,E1 -7041.395,E2 -7041.395} C_VEL
LIN {X 0,Y 481.67,Z 361.487,A -85,B 0,C 180,E1 -7044.114,E2 -7044.114} C_VEL
LIN {X 0,Y 481.746,Z 361.467,A -85,B 0,C 180,E1 -7047.141,E2 -7047.141} C_VEL
LIN {X 0,Y 481.673,Z 361.484,A -85,B 0,C 180,E1 -7049.742,E2 -7049.742} C_VEL
LIN {X 0,Y 481.668,Z 361.485,A -85,B 0,C 180,E1 -7052.675,E2 -7052.675} C_VEL
LIN {X 0,Y 481.638,Z 361.489,A -85,B 0,C 180,E1 -7055.71,E2 -7055.71} C_VEL
LIN {X 0,Y 481.711,Z 361.478,A -85,B 0,C 180,E1 -7059.355,E2 -7059.355} C_VEL
LIN {X 0,Y 481.671,Z 361.485,A -85,B 0,C 180,E1 -7062.159,E2 -7062.159} C_VEL
LIN {X 0,Y 481.658,Z 361.489,A -85,B 0,C 180,E1 -7064.458,E2 -7064.458} C_VEL
LIN {X 0,Y 481.648,Z 361.495,A -85,B 0,C 180,E1 -7067.841,E2 -7067.841} C_VEL
LIN {X 0,Y 481.72,Z 361.478,A -85,B 0,C 180,E1 -7070.646,E2 -7070.646} C_VEL
LIN {X 0,Y 481.644,Z 361.489,A -85,B 0,C 180,E1 -7074.292,E2 -7074.292} C_VEL
LIN {X 0,Y 481.674,Z 361.486,A -85,B 0,C 180,E1 -7077.327,E2 -7077.327} C_VEL
LIN {X 0,Y 481.764,Z 361.65,A -85,B 0,C 180,E1 -7080.878,E2 -7080.878} C_VEL
LIN {X 0,Y 482.724,Z 367.427,A -85,B 0,C 180,E1 -7082.233,E2 -7082.233} C_VEL
LIN {X 0,Y 482.46,Z 377.984,A -85,B 0,C 180,E1 -7084.536,E2 -7084.536} C_VEL
LIN {X 0,Y 485.12,Z 391.665,A -85,B 0,C 180,E1 -7084.846,E2 -7084.846} C_VEL
LIN {X 0,Y 485.019,Z 403.879,A -85,B 0,C 180,E1 -7085.029,E2 -7085.029} C_VEL
LIN {X 0,Y 484.305,Z 409.728,A -85,B 0,C 180,E1 -7085.091,E2 -7085.091} C_VEL
LIN {X 0,Y 478.56,Z 428.723,A -85,B 0,C 180,E1 -7085.17,E2 -7085.17} C_VEL
LIN {X 0,Y 477.937,Z 434.567,A -85,B 0,C 180,E1 -7085.237,E2 -7085.237} C_VEL
LIN {X 0,Y 477.545,Z 484.954,A -85,B 0,C 180,E1 -7086.025,E2 -7086.025} C_VEL
LIN {X 0,Y 477.281,Z 497.639,A -85,B 0,C 180,E1 -7086.386,E2 -7086.386} C_VEL
LIN {X 0,Y 476.952,Z 509.882,A -85,B 0,C 180,E1 -7086.901,E2 -7086.901} C_VEL
LIN {X 0,Y 476.592,Z 521.641,A -85,B 0,C 180,E1 -7087.57,E2 -7087.57} C_VEL
LIN {X 0,Y 476.141,Z 533.141,A -85,B 0,C 180,E1 -7088.421,E2 -7088.421} C_VEL
LIN {X 0,Y 475.663,Z 543.163,A -85,B 0,C 180,E1 -7089.344,E2 -7089.344} C_VEL
LIN {X 0,Y 475.203,Z 551.998,A -85,B 0,C 180,E1 -7090.339,E2 -7090.339} C_VEL
LIN {X 0,Y 474.77,Z 561.034,A -85,B 0,C 180,E1 -7091.593,E2 -7091.593} C_VEL
LIN {X 0,Y 474.44,Z 569.025,A -85,B 0,C 180,E1 -7092.989,E2 -7092.989} C_VEL
LIN {X 0,Y 474.154,Z 575.636,A -85,B 0,C 180,E1 -7094.462,E2 -7094.462} C_VEL
LIN {X 0,Y 473.948,Z 580.345,A -85,B 0,C 180,E1 -7095.838,E2 -7095.838} C_VEL
LIN {X 0,Y 473.858,Z 583.693,A -85,B 0,C 180,E1 -7097.146,E2 -7097.146} C_VEL
LIN {X 0,Y 473.821,Z 585.698,A -85,B 0,C 180,E1 -7098.226,E2 -7098.226} C_VEL
LIN {X 0,Y 473.707,Z 587.392,A -85,B 0,C 180,E1 -7099.745,E2 -7099.745} C_VEL
LIN {X 0,Y 473.728,Z 587.768,A -85,B 0,C 180,E1 -7101.469,E2 -7101.469} C_VEL
LIN {X 0,Y 473.752,Z 587.379,A -85,B 0,C 180,E1 -7102.328,E2 -7102.328} C_VEL
LIN {X 0,Y 473.836,Z 586.028,A -85,B 0,C 180,E1 -7103.598,E2 -7103.598} C_VEL
LIN {X 0,Y 473.818,Z 582.758,A -85,B 0,C 180,E1 -7105.321,E2 -7105.321} C_VEL
LIN {X 0,Y 474.029,Z 579.159,A -85,B 0,C 180,E1 -7106.6,E2 -7106.6} C_VEL
LIN {X 0,Y 474.119,Z 574.485,A -85,B 0,C 180,E1 -7107.876,E2 -7107.876} C_VEL
LIN {X 0,Y 474.455,Z 567.467,A -85,B 0,C 180,E1 -7109.363,E2 -7109.363} C_VEL
LIN {X 0,Y 474.775,Z 559.861,A -85,B 0,C 180,E1 -7110.636,E2 -7110.636} C_VEL
LIN {X 0,Y 475.215,Z 550.337,A -85,B 0,C 180,E1 -7111.907,E2 -7111.907} C_VEL
LIN {X 0,Y 475.58,Z 540.543,A -85,B 0,C 180,E1 -7112.965,E2 -7112.965} C_VEL
LIN {X 0,Y 476.06,Z 529.48,A -85,B 0,C 180,E1 -7113.915,E2 -7113.915} C_VEL
LIN {X 0,Y 476.532,Z 518.655,A -85,B 0,C 180,E1 -7114.653,E2 -7114.653} C_VEL
LIN {X 0,Y 476.865,Z 506.745,A -85,B 0,C 180,E1 -7115.285,E2 -7115.285} C_VEL
LIN {X 0,Y 477.158,Z 494.477,A -85,B 0,C 180,E1 -7115.759,E2 -7115.759} C_VEL
LIN {X 0,Y 477.4,Z 481.761,A -85,B 0,C 180,E1 -7116.074,E2 -7116.074} C_VEL
LIN {X 0,Y 478.135,Z 390.583,A -85,B 0,C 180,E1 -7117.453,E2 -7117.453} C_VEL
LIN {X 0,Y 475.435,Z 377.904,A -85,B 0,C 180,E1 -7117.763,E2 -7117.763} C_VEL
LIN {X 0,Y 475.621,Z 368.724,A -85,B 0,C 180,E1 -7119.783,E2 -7119.783} C_VEL
LIN {X 0,Y 474.771,Z 362.348,A -85,B 0,C 180,E1 -7121.257,E2 -7121.257} C_VEL
LIN {X 0,Y 474.654,Z 362.362,A -85,B 0,C 180,E1 -7124.578,E2 -7124.578} C_VEL
LIN {X 0,Y 474.653,Z 362.356,A -85,B 0,C 180,E1 -7127.225,E2 -7127.225} C_VEL
LIN {X 0,Y 474.659,Z 362.358,A -85,B 0,C 180,E1 -7129.91,E2 -7129.91} C_VEL
LIN {X 0,Y 474.64,Z 362.358,A -85,B 0,C 180,E1 -7133.358,E2 -7133.358} C_VEL
LIN {X 0,Y 474.664,Z 362.361,A -85,B 0,C 180,E1 -7136.371,E2 -7136.371} C_VEL
LIN {X 0,Y 474.632,Z 362.36,A -85,B 0,C 180,E1 -7139.25,E2 -7139.25} C_VEL
LIN {X 0,Y 474.617,Z 362.365,A -85,B 0,C 180,E1 -7142.43,E2 -7142.43} C_VEL
LIN {X 0,Y 474.621,Z 362.362,A -85,B 0,C 180,E1 -7145.469,E2 -7145.469} C_VEL
LIN {X 0,Y 474.612,Z 362.365,A -85,B 0,C 180,E1 -7148.456,E2 -7148.456} C_VEL
LIN {X 0,Y 474.626,Z 362.361,A -85,B 0,C 180,E1 -7150.958,E2 -7150.958} C_VEL
LIN {X 0,Y 474.607,Z 362.368,A -85,B 0,C 180,E1 -7154.104,E2 -7154.104} C_VEL
LIN {X 0,Y 474.649,Z 362.359,A -85,B 0,C 180,E1 -7157.069,E2 -7157.069} C_VEL
LIN {X 0,Y 474.665,Z 362.357,A -85,B 0,C 180,E1 -7160.456,E2 -7160.456} C_VEL
LIN {X 0,Y 474.587,Z 362.369,A -85,B 0,C 180,E1 -7163.676,E2 -7163.676} C_VEL
LIN {X 0,Y 474.638,Z 362.36,A -85,B 0,C 180,E1 -7166.779,E2 -7166.779} C_VEL
LIN {X 0,Y 474.6,Z 362.369,A -85,B 0,C 180,E1 -7169.769,E2 -7169.769} C_VEL
LIN {X 0,Y 474.708,Z 362.352,A -85,B 0,C 180,E1 -7172.68,E2 -7172.68} C_VEL
LIN {X 0,Y 474.656,Z 362.361,A -85,B 0,C 180,E1 -7175.507,E2 -7175.507} C_VEL
LIN {X 0,Y 474.669,Z 362.358,A -85,B 0,C 180,E1 -7179.185,E2 -7179.185} C_VEL
LIN {X 0,Y 474.649,Z 362.361,A -85,B 0,C 180,E1 -7181.884,E2 -7181.884} C_VEL
LIN {X 0,Y 474.692,Z 362.354,A -85,B 0,C 180,E1 -7184.544,E2 -7184.544} C_VEL
LIN {X 0,Y 474.73,Z 362.349,A -85,B 0,C 180,E1 -7188.038,E2 -7188.038} C_VEL
LIN {X 0,Y 474.721,Z 362.353,A -85,B 0,C 180,E1 -7191.486,E2 -7191.486} C_VEL
LIN {X 0,Y 474.771,Z 362.344,A -85,B 0,C 180,E1 -7194.052,E2 -7194.052} C_VEL
LIN {X 0,Y 474.887,Z 362.332,A -85,B 0,C 180,E1 -7197.455,E2 -7197.455} C_VEL
LIN {X 0,Y 474.869,Z 362.334,A -85,B 0,C 180,E1 -7200.848,E2 -7200.848} C_VEL
LIN {X 0,Y 474.887,Z 362.332,A -85,B 0,C 180,E1 -7202.544,E2 -7202.544} C_VEL
LIN {X 0,Y 474.775,Z 362.343,A -85,B 0,C 180,E1 -7205.947,E2 -7205.947} C_VEL
LIN {X 0,Y 474.72,Z 362.354,A -85,B 0,C 180,E1 -7208.513,E2 -7208.513} C_VEL
LIN {X 0,Y 474.73,Z 362.349,A -85,B 0,C 180,E1 -7211.962,E2 -7211.962} C_VEL
LIN {X 0,Y 474.691,Z 362.354,A -85,B 0,C 180,E1 -7215.456,E2 -7215.456} C_VEL
LIN {X 0,Y 474.657,Z 362.359,A -85,B 0,C 180,E1 -7219.01,E2 -7219.01} C_VEL
LIN {X 0,Y 474.6,Z 362.365,A -85,B 0,C 180,E1 -7221.728,E2 -7221.728} C_VEL
LIN {X 0,Y 474.654,Z 362.362,A -85,B 0,C 180,E1 -7224.493,E2 -7224.493} C_VEL
LIN {X 0,Y 474.691,Z 362.354,A -85,B 0,C 180,E1 -7227.339,E2 -7227.339} C_VEL
LIN {X 0,Y 474.598,Z 362.366,A -85,B 0,C 180,E1 -7230.811,E2 -7230.811} C_VEL
LIN {X 0,Y 474.632,Z 362.363,A -85,B 0,C 180,E1 -7233.985,E2 -7233.985} C_VEL
LIN {X 0,Y 474.57,Z 362.369,A -85,B 0,C 180,E1 -7236.901,E2 -7236.901} C_VEL
LIN {X 0,Y 474.645,Z 362.36,A -85,B 0,C 180,E1 -7239.652,E2 -7239.652} C_VEL
LIN {X 0,Y 474.646,Z 362.359,A -85,B 0,C 180,E1 -7242.931,E2 -7242.931} C_VEL
LIN {X 0,Y 474.605,Z 362.368,A -85,B 0,C 180,E1 -7245.896,E2 -7245.896} C_VEL
LIN {X 0,Y 474.624,Z 362.36,A -85,B 0,C 180,E1 -7249.041,E2 -7249.041} C_VEL
LIN {X 0,Y 474.608,Z 362.366,A -85,B 0,C 180,E1 -7251.705,E2 -7251.705} C_VEL
LIN {X 0,Y 474.628,Z 362.36,A -85,B 0,C 180,E1 -7254.727,E2 -7254.727} C_VEL
LIN {X 0,Y 474.637,Z 362.364,A -85,B 0,C 180,E1 -7257.789,E2 -7257.789} C_VEL
LIN {X 0,Y 474.632,Z 362.361,A -85,B 0,C 180,E1 -7260.883,E2 -7260.883} C_VEL
LIN {X 0,Y 474.708,Z 362.409,A -85,B 0,C 180,E1 -7263.66,E2 -7263.66} C_VEL
LIN {X 0,Y 476.991,Z 374.688,A -85,B 0,C 180,E1 -7265.879,E2 -7265.879} C_VEL
LIN {X 0,Y 476.263,Z 392.185,A -85,B 0,C 180,E1 -7268.806,E2 -7268.806} C_VEL
LIN {X 0,Y 475.569,Z 411.018,A -85,B 0,C 180,E1 -7271.921,E2 -7271.921} C_VEL
LIN {X 0,Y 475.26,Z 419.163,A -85,B 0,C 180,E1 -7273.257,E2 -7273.257} C_VEL
LIN {X 0,Y 477.948,Z 437.082,A -85,B 0,C 180,E1 -7273.627,E2 -7273.627} C_VEL
LIN {X 0,Y 477.344,Z 527.953,A -85,B 0,C 180,E1 -7275.015,E2 -7275.015} C_VEL
LIN {X 0,Y 476.976,Z 541.198,A -85,B 0,C 180,E1 -7275.385,E2 -7275.385} C_VEL
LIN {X 0,Y 476.539,Z 553.931,A -85,B 0,C 180,E1 -7275.916,E2 -7275.916} C_VEL
LIN {X 0,Y 476.105,Z 565.25,A -85,B 0,C 180,E1 -7276.557,E2 -7276.557} C_VEL
LIN {X 0,Y 475.603,Z 576.711,A -85,B 0,C 180,E1 -7277.392,E2 -7277.392} C_VEL
LIN {X 0,Y 475.198,Z 587.474,A -85,B 0,C 180,E1 -7278.375,E2 -7278.375} C_VEL
LIN {X 0,Y 474.779,Z 596.076,A -85,B 0,C 180,E1 -7279.337,E2 -7279.337} C_VEL
LIN {X 0,Y 474.436,Z 604.011,A -85,B 0,C 180,E1 -7280.407,E2 -7280.407} C_VEL
LIN {X 0,Y 474.151,Z 611.762,A -85,B 0,C 180,E1 -7281.691,E2 -7281.691} C_VEL
LIN {X 0,Y 473.934,Z 618.9,A -85,B 0,C 180,E1 -7283.187,E2 -7283.187} C_VEL
LIN {X 0,Y 473.846,Z 623.651,A -85,B 0,C 180,E1 -7284.468,E2 -7284.468} C_VEL
LIN {X 0,Y 473.748,Z 627.278,A -85,B 0,C 180,E1 -7285.746,E2 -7285.746} C_VEL
LIN {X 0,Y 473.801,Z 629.154,A -85,B 0,C 180,E1 -7286.599,E2 -7286.599} C_VEL
LIN {X 0,Y 473.761,Z 630.556,A -85,B 0,C 180,E1 -7287.449,E2 -7287.449} C_VEL
LIN {X 0,Y 473.756,Z 631.555,A -85,B 0,C 180,E1 -7288.3,E2 -7288.3} C_VEL
LIN {X 0,Y 473.672,Z 632.377,A -85,B 0,C 180,E1 -7290,E2 -7290} C_VEL
LIN {X 0,Y 473.756,Z 631.548,A -85,B 0,C 180,E1 -7291.7,E2 -7291.7} C_VEL
LIN {X 0,Y 473.761,Z 630.546,A -85,B 0,C 180,E1 -7292.551,E2 -7292.551} C_VEL
LIN {X 0,Y 473.801,Z 629.142,A -85,B 0,C 180,E1 -7293.401,E2 -7293.401} C_VEL
LIN {X 0,Y 473.763,Z 626.187,A -85,B 0,C 180,E1 -7294.68,E2 -7294.68} C_VEL
LIN {X 0,Y 473.834,Z 622.195,A -85,B 0,C 180,E1 -7295.959,E2 -7295.959} C_VEL
LIN {X 0,Y 474.015,Z 616.063,A -85,B 0,C 180,E1 -7297.454,E2 -7297.454} C_VEL
LIN {X 0,Y 474.228,Z 609.365,A -85,B 0,C 180,E1 -7298.737,E2 -7298.737} C_VEL
LIN {X 0,Y 474.541,Z 601.067,A -85,B 0,C 180,E1 -7300.021,E2 -7300.021} C_VEL
LIN {X 0,Y 474.986,Z 592.58,A -85,B 0,C 180,E1 -7301.09,E2 -7301.09} C_VEL
LIN {X 0,Y 475.458,Z 582.39,A -85,B 0,C 180,E1 -7302.133,E2 -7302.133} C_VEL
LIN {X 0,Y 475.813,Z 572.034,A -85,B 0,C 180,E1 -7302.995,E2 -7302.995} C_VEL
LIN {X 0,Y 476.343,Z 560.427,A -85,B 0,C 180,E1 -7303.763,E2 -7303.763} C_VEL
LIN {X 0,Y 476.788,Z 548.896,A -85,B 0,C 180,E1 -7304.348,E2 -7304.348} C_VEL
LIN {X 0,Y 477.217,Z 535.667,A -85,B 0,C 180,E1 -7304.826,E2 -7304.826} C_VEL
LIN {X 0,Y 477.481,Z 522.862,A -85,B 0,C 180,E1 -7305.117,E2 -7305.117} C_VEL
LIN {X 0,Y 478.064,Z 437.443,A -85,B 0,C 180,E1 -7306.415,E2 -7306.415} C_VEL
LIN {X 0,Y 475.318,Z 419.003,A -85,B 0,C 180,E1 -7306.813,E2 -7306.813} C_VEL
LIN {X 0,Y 476.079,Z 399.434,A -85,B 0,C 180,E1 -7310.073,E2 -7310.073} C_VEL
LIN {X 0,Y 476.976,Z 379.551,A -85,B 0,C 180,E1 -7313.442,E2 -7313.442} C_VEL
LIN {X 0,Y 477.064,Z 374.252,A -85,B 0,C 180,E1 -7314.361,E2 -7314.361} C_VEL
LIN {X 0,Y 474.818,Z 362.99,A -85,B 0,C 180,E1 -7316.48,E2 -7316.48} C_VEL
LIN {X 0,Y 474.691,Z 362.358,A -85,B 0,C 180,E1 -7316.606,E2 -7316.606} C_VEL
LIN {X 0,Y 474.63,Z 362.361,A -85,B 0,C 180,E1 -7319.251,E2 -7319.251} C_VEL
LIN {X 0,Y 474.616,Z 362.365,A -85,B 0,C 180,E1 -7322.43,E2 -7322.43} C_VEL
LIN {X 0,Y 474.618,Z 362.364,A -85,B 0,C 180,E1 -7325.47,E2 -7325.47} C_VEL
LIN {X 0,Y 474.609,Z 362.363,A -85,B 0,C 180,E1 -7328.456,E2 -7328.456} C_VEL
LIN {X 0,Y 474.624,Z 362.359,A -85,B 0,C 180,E1 -7330.959,E2 -7330.959} C_VEL
LIN {X 0,Y 474.605,Z 362.364,A -85,B 0,C 180,E1 -7334.104,E2 -7334.104} C_VEL
LIN {X 0,Y 474.646,Z 362.356,A -85,B 0,C 180,E1 -7337.069,E2 -7337.069} C_VEL
LIN {X 0,Y 474.663,Z 362.354,A -85,B 0,C 180,E1 -7340.456,E2 -7340.456} C_VEL
LIN {X 0,Y 474.587,Z 362.37,A -85,B 0,C 180,E1 -7343.676,E2 -7343.676} C_VEL
LIN {X 0,Y 474.636,Z 362.359,A -85,B 0,C 180,E1 -7346.779,E2 -7346.779} C_VEL
LIN {X 0,Y 474.607,Z 362.365,A -85,B 0,C 180,E1 -7349.77,E2 -7349.77} C_VEL
LIN {X 0,Y 474.707,Z 362.349,A -85,B 0,C 180,E1 -7352.681,E2 -7352.681} C_VEL
LIN {X 0,Y 474.654,Z 362.351,A -85,B 0,C 180,E1 -7355.507,E2 -7355.507} C_VEL
LIN {X 0,Y 474.663,Z 362.362,A -85,B 0,C 180,E1 -7359.185,E2 -7359.185} C_VEL
LIN {X 0,Y 474.648,Z 362.357,A -85,B 0,C 180,E1 -7361.884,E2 -7361.884} C_VEL
LIN {X 0,Y 474.691,Z 362.351,A -85,B 0,C 180,E1 -7364.544,E2 -7364.544} C_VEL
LIN {X 0,Y 474.73,Z 362.346,A -85,B 0,C 180,E1 -7368.038,E2 -7368.038} C_VEL
LIN {X 0,Y 474.72,Z 362.35,A -85,B 0,C 180,E1 -7371.487,E2 -7371.487} C_VEL
LIN {X 0,Y 474.771,Z 362.338,A -85,B 0,C 180,E1 -7374.052,E2 -7374.052} C_VEL
LIN {X 0,Y 474.887,Z 362.327,A -85,B 0,C 180,E1 -7377.456,E2 -7377.456} C_VEL
LIN {X 0,Y 474.869,Z 362.337,A -85,B 0,C 180,E1 -7380.848,E2 -7380.848} C_VEL
LIN {X 0,Y 474.887,Z 362.331,A -85,B 0,C 180,E1 -7382.545,E2 -7382.545} C_VEL
LIN {X 0,Y 474.771,Z 362.342,A -85,B 0,C 180,E1 -7385.948,E2 -7385.948} C_VEL
LIN {X 0,Y 474.72,Z 362.35,A -85,B 0,C 180,E1 -7388.514,E2 -7388.514} C_VEL
LIN {X 0,Y 474.697,Z 362.351,A -85,B 0,C 180,E1 -7391.963,E2 -7391.963} C_VEL
LIN {X 0,Y 474.692,Z 362.351,A -85,B 0,C 180,E1 -7395.456,E2 -7395.456} C_VEL
LIN {X 0,Y 474.658,Z 362.357,A -85,B 0,C 180,E1 -7399.011,E2 -7399.011} C_VEL
LIN {X 0,Y 474.582,Z 362.364,A -85,B 0,C 180,E1 -7401.73,E2 -7401.73} C_VEL
LIN {X 0,Y 474.652,Z 362.357,A -85,B 0,C 180,E1 -7404.494,E2 -7404.494} C_VEL
LIN {X 0,Y 474.693,Z 362.345,A -85,B 0,C 180,E1 -7407.34,E2 -7407.34} C_VEL
LIN {X 0,Y 474.599,Z 362.362,A -85,B 0,C 180,E1 -7410.811,E2 -7410.811} C_VEL
LIN {X 0,Y 474.634,Z 362.364,A -85,B 0,C 180,E1 -7413.985,E2 -7413.985} C_VEL
LIN {X 0,Y 474.571,Z 362.367,A -85,B 0,C 180,E1 -7416.901,E2 -7416.901} C_VEL
LIN {X 0,Y 474.647,Z 362.36,A -85,B 0,C 180,E1 -7419.652,E2 -7419.652} C_VEL
LIN {X 0,Y 474.649,Z 362.357,A -85,B 0,C 180,E1 -7422.931,E2 -7422.931} C_VEL
LIN {X 0,Y 474.607,Z 362.368,A -85,B 0,C 180,E1 -7425.896,E2 -7425.896} C_VEL
LIN {X 0,Y 474.64,Z 362.361,A -85,B 0,C 180,E1 -7429.04,E2 -7429.04} C_VEL
LIN {X 0,Y 474.62,Z 362.368,A -85,B 0,C 180,E1 -7431.703,E2 -7431.703} C_VEL
LIN {X 0,Y 474.631,Z 362.361,A -85,B 0,C 180,E1 -7434.727,E2 -7434.727} C_VEL
LIN {X 0,Y 474.638,Z 362.365,A -85,B 0,C 180,E1 -7437.789,E2 -7437.789} C_VEL
LIN {X 0,Y 474.722,Z 362.476,A -85,B 0,C 180,E1 -7440.664,E2 -7440.664} C_VEL
LIN {X 0,Y 475.792,Z 369.849,A -85,B 0,C 180,E1 -7442.409,E2 -7442.409} C_VEL
LIN {X 0,Y 475.532,Z 378.142,A -85,B 0,C 180,E1 -7444.261,E2 -7444.261} C_VEL
LIN {X 0,Y 478.319,Z 391.479,A -85,B 0,C 180,E1 -7444.585,E2 -7444.585} C_VEL
LIN {X 0,Y 477.937,Z 434.567,A -85,B 0,C 180,E1 -7445.237,E2 -7445.237} C_VEL
LIN {X 0,Y 477.316,Z 440.411,A -85,B 0,C 180,E1 -7445.304,E2 -7445.304} C_VEL
LIN {X 0,Y 471.622,Z 459.413,A -85,B 0,C 180,E1 -7445.386,E2 -7445.386} C_VEL
LIN {X 0,Y 470.941,Z 465.261,A -85,B 0,C 180,E1 -7445.452,E2 -7445.452} C_VEL
LIN {X 0,Y 470.705,Z 486.601,A -85,B 0,C 180,E1 -7445.815,E2 -7445.815} C_VEL
LIN {X 0,Y 470.446,Z 499.687,A -85,B 0,C 180,E1 -7446.213,E2 -7446.213} C_VEL
LIN {X 0,Y 470.049,Z 512.225,A -85,B 0,C 180,E1 -7446.775,E2 -7446.775} C_VEL
LIN {X 0,Y 469.694,Z 523.455,A -85,B 0,C 180,E1 -7447.455,E2 -7447.455} C_VEL
LIN {X 0,Y 469.148,Z 535.185,A -85,B 0,C 180,E1 -7448.359,E2 -7448.359} C_VEL
LIN {X 0,Y 468.603,Z 545.519,A -85,B 0,C 180,E1 -7449.363,E2 -7449.363} C_VEL
LIN {X 0,Y 468.124,Z 554.814,A -85,B 0,C 180,E1 -7450.486,E2 -7450.486} C_VEL
LIN {X 0,Y 467.734,Z 562.429,A -85,B 0,C 180,E1 -7451.607,E2 -7451.607} C_VEL
LIN {X 0,Y 467.395,Z 569.855,A -85,B 0,C 180,E1 -7452.95,E2 -7452.95} C_VEL
LIN {X 0,Y 467.098,Z 576.003,A -85,B 0,C 180,E1 -7454.357,E2 -7454.357} C_VEL
LIN {X 0,Y 466.906,Z 580.322,A -85,B 0,C 180,E1 -7455.62,E2 -7455.62} C_VEL
LIN {X 0,Y 466.789,Z 583.771,A -85,B 0,C 180,E1 -7456.948,E2 -7456.948} C_VEL
LIN {X 0,Y 466.745,Z 586.023,A -85,B 0,C 180,E1 -7458.166,E2 -7458.166} C_VEL
LIN {X 0,Y 466.637,Z 587.64,A -85,B 0,C 180,E1 -7459.588,E2 -7459.588} C_VEL
LIN {X 0,Y 466.582,Z 588.086,A -85,B 0,C 180,E1 -7460.463,E2 -7460.463} C_VEL
LIN {X 0,Y 466.635,Z 588.125,A -85,B 0,C 180,E1 -7461.338,E2 -7461.338} C_VEL
LIN {X 0,Y 466.705,Z 587.051,A -85,B 0,C 180,E1 -7463.081,E2 -7463.081} C_VEL
LIN {X 0,Y 466.765,Z 585.883,A -85,B 0,C 180,E1 -7463.95,E2 -7463.95} C_VEL
LIN {X 0,Y 466.741,Z 584.313,A -85,B 0,C 180,E1 -7464.817,E2 -7464.817} C_VEL
LIN {X 0,Y 466.892,Z 581.153,A -85,B 0,C 180,E1 -7466.116,E2 -7466.116} C_VEL
LIN {X 0,Y 466.986,Z 576.957,A -85,B 0,C 180,E1 -7467.412,E2 -7467.412} C_VEL
LIN {X 0,Y 467.258,Z 570.596,A -85,B 0,C 180,E1 -7468.923,E2 -7468.923} C_VEL
LIN {X 0,Y 467.6,Z 563.649,A -85,B 0,C 180,E1 -7470.215,E2 -7470.215} C_VEL
